LIN {X 0,Y 540.367,Z 1010.165,A -85,B 0,C 180,E1 3978.151,E2 3978.151} C_VEL
LIN {X 0,Y 538.15,Z 995.311,A -85,B 0,C 180,E1 3978.449,E2 3978.449} C_VEL
LIN {X 0,Y 536.475,Z 989.03,A -85,B 0,C 180,E1 3978.66,E2 3978.66} C_VEL
LIN {X 0,Y 536.148,Z 989.03,A -85,B 0,C 180,E1 3984.971,E2 3984.971} C_VEL
LIN {X 0,Y 536.089,Z 989.03,A -85,B 0,C 180,E1 3990.441,E2 3990.441} C_VEL
LIN {X 0,Y 536.003,Z 989.03,A -85,B 0,C 180,E1 3996.241,E2 3996.241} C_VEL
LIN {X 0,Y 535.964,Z 989.03,A -85,B 0,C 180,E1 4002.507,E2 4002.507} C_VEL
LIN {X 0,Y 536.056,Z 989.03,A -85,B 0,C 180,E1 4007.493,E2 4007.493} C_VEL
LIN {X 0,Y 536.117,Z 989.03,A -85,B 0,C 180,E1 4013.761,E2 4013.761} C_VEL
LIN {X 0,Y 536.077,Z 989.03,A -85,B 0,C 180,E1 4019.552,E2 4019.552} C_VEL
LIN {X 0,Y 536.133,Z 989.03,A -85,B 0,C 180,E1 4020.914,E2 4020.914} C_VEL
LIN {X 0,Y 544.829,Z 1011.912,A -85,B 0,C 180,E1 4021.779,E2 4021.779} C_VEL
LIN {X 0,Y 544.168,Z 1050.277,A -85,B 0,C 180,E1 4022.566,E2 4022.566} C_VEL
LIN {X 0,Y 543.022,Z 1087.066,A -85,B 0,C 180,E1 4023.969,E2 4023.969} C_VEL
LIN {X 0,Y 541.475,Z 1121.1,A -85,B 0,C 180,E1 4025.943,E2 4025.943} C_VEL
LIN {X 0,Y 539.972,Z 1152.521,A -85,B 0,C 180,E1 4028.483,E2 4028.483} C_VEL
LIN {X 0,Y 538.584,Z 1181.234,A -85,B 0,C 180,E1 4031.623,E2 4031.623} C_VEL
LIN {X 0,Y 537.575,Z 1204.956,A -85,B 0,C 180,E1 4035.155,E2 4035.155} C_VEL
LIN {X 0,Y 537.021,Z 1223.191,A -85,B 0,C 180,E1 4038.924,E2 4038.924} C_VEL
LIN {X 0,Y 536.82,Z 1235.502,A -85,B 0,C 180,E1 4042.73,E2 4042.73} C_VEL
LIN {X 0,Y 536.779,Z 1242.723,A -85,B 0,C 180,E1 4046.774,E2 4046.774} C_VEL
LIN {X 0,Y 536.69,Z 1244.497,A -85,B 0,C 180,E1 4049.997,E2 4049.997} C_VEL
LIN {X 0,Y 536.816,Z 1241.65,A -85,B 0,C 180,E1 4054.01,E2 4054.01} C_VEL
LIN {X 0,Y 536.89,Z 1233.07,A -85,B 0,C 180,E1 4058.076,E2 4058.076} C_VEL
LIN {X 0,Y 537.166,Z 1219.982,A -85,B 0,C 180,E1 4061.749,E2 4061.749} C_VEL
LIN {X 0,Y 537.78,Z 1200.841,A -85,B 0,C 180,E1 4065.458,E2 4065.458} C_VEL
LIN {X 0,Y 538.787,Z 1177.187,A -85,B 0,C 180,E1 4068.786,E2 4068.786} C_VEL
LIN {X 0,Y 540.151,Z 1149.395,A -85,B 0,C 180,E1 4071.717,E2 4071.717} C_VEL
LIN {X 0,Y 541.704,Z 1116.776,A -85,B 0,C 180,E1 4074.258,E2 4074.258} C_VEL
LIN {X 0,Y 543.1,Z 1082.588,A -85,B 0,C 180,E1 4076.148,E2 4076.148} C_VEL
LIN {X 0,Y 544.272,Z 1045.483,A -85,B 0,C 180,E1 4077.481,E2 4077.481} C_VEL
LIN {X 0,Y 544.242,Z 1008.876,A -85,B 0,C 180,E1 4078.209,E2 4078.209} C_VEL
LIN {X 0,Y 536.279,Z 989.03,A -85,B 0,C 180,E1 4079.036,E2 4079.036} C_VEL
LIN {X 0,Y 536.021,Z 989.03,A -85,B 0,C 180,E1 4085.277,E2 4085.277} C_VEL
LIN {X 0,Y 535.953,Z 989.03,A -85,B 0,C 180,E1 4090.522,E2 4090.522} C_VEL
LIN {X 0,Y 536.032,Z 989.03,A -85,B 0,C 180,E1 4097.046,E2 4097.046} C_VEL
LIN {X 0,Y 536.16,Z 989.03,A -85,B 0,C 180,E1 4102.001,E2 4102.001} C_VEL
LIN {X 0,Y 536.064,Z 989.03,A -85,B 0,C 180,E1 4107.669,E2 4107.669} C_VEL
LIN {X 0,Y 536.162,Z 989.03,A -85,B 0,C 180,E1 4113.238,E2 4113.238} C_VEL
LIN {X 0,Y 536.256,Z 989.03,A -85,B 0,C 180,E1 4118.544,E2 4118.544} C_VEL
LIN {X 0,Y 536.371,Z 989.03,A -85,B 0,C 180,E1 4123.661,E2 4123.661} C_VEL
LIN {X 0,Y 536.376,Z 989.03,A -85,B 0,C 180,E1 4128.643,E2 4128.643} C_VEL
LIN {X 0,Y 536.424,Z 989.03,A -85,B 0,C 180,E1 4133.54,E2 4133.54} C_VEL
LIN {X 0,Y 536.402,Z 989.03,A -85,B 0,C 180,E1 4138.388,E2 4138.388} C_VEL
LIN {X 0,Y 536.458,Z 989.03,A -85,B 0,C 180,E1 4143.225,E2 4143.225} C_VEL
LIN {X 0,Y 536.344,Z 989.03,A -85,B 0,C 180,E1 4148.087,E2 4148.087} C_VEL
LIN {X 0,Y 536.321,Z 989.03,A -85,B 0,C 180,E1 4153.008,E2 4153.008} C_VEL
LIN {X 0,Y 536.256,Z 989.03,A -85,B 0,C 180,E1 4158.031,E2 4158.031} C_VEL
LIN {X 0,Y 536.189,Z 989.03,A -85,B 0,C 180,E1 4163.203,E2 4163.203} C_VEL
LIN {X 0,Y 536.17,Z 989.03,A -85,B 0,C 180,E1 4166.745,E2 4166.745} C_VEL
LIN {X 0,Y 533.647,Z 989.03,A -85,B 0,C 180,E1 4168.125,E2 4168.125} C_VEL
LIN {X 0,Y 528.17,Z 989.03,A -85,B 0,C 180,E1 4170.192,E2 4170.192} C_VEL
LIN {X 0,Y 528.081,Z 989.03,A -85,B 0,C 180,E1 4170.431,E2 4170.431} C_VEL
LIN {X 0,Y 528.183,Z 989.03,A -85,B 0,C 180,E1 4176.877,E2 4176.877} C_VEL
LIN {X 0,Y 528.102,Z 989.03,A -85,B 0,C 180,E1 4182.021,E2 4182.021} C_VEL
LIN {X 0,Y 527.988,Z 989.03,A -85,B 0,C 180,E1 4187.993,E2 4187.993} C_VEL
LIN {X 0,Y 528.102,Z 989.11,A -85,B 0,C 180,E1 4193.2,E2 4193.2} C_VEL
LIN {X 0,Y 531.272,Z 996.761,A -85,B 0,C 180,E1 4194.015,E2 4194.015} C_VEL
LIN {X 0,Y 534.684,Z 1001.319,A -85,B 0,C 180,E1 4194.927,E2 4194.927} C_VEL
LIN {X 0,Y 536.379,Z 1002.647,A -85,B 0,C 180,E1 4195.518,E2 4195.518} C_VEL
LIN {X 0,Y 536.746,Z 1007.356,A -85,B 0,C 180,E1 4196.014,E2 4196.014} C_VEL
LIN {X 0,Y 540.769,Z 1015.949,A -85,B 0,C 180,E1 4196.435,E2 4196.435} C_VEL
LIN {X 0,Y 540.154,Z 1080.881,A -85,B 0,C 180,E1 4197.563,E2 4197.563} C_VEL
LIN {X 0,Y 538.764,Z 1119.195,A -85,B 0,C 180,E1 4198.853,E2 4198.853} C_VEL
LIN {X 0,Y 536.801,Z 1156.353,A -85,B 0,C 180,E1 4200.759,E2 4200.759} C_VEL
LIN {X 0,Y 534.581,Z 1192.701,A -85,B 0,C 180,E1 4203.38,E2 4203.38} C_VEL
LIN {X 0,Y 532.599,Z 1224.03,A -85,B 0,C 180,E1 4206.412,E2 4206.412} C_VEL
LIN {X 0,Y 530.966,Z 1251.131,A -85,B 0,C 180,E1 4209.821,E2 4209.821} C_VEL
LIN {X 0,Y 529.76,Z 1274.259,A -85,B 0,C 180,E1 4213.666,E2 4213.666} C_VEL
LIN {X 0,Y 529.131,Z 1292.024,A -85,B 0,C 180,E1 4217.652,E2 4217.652} C_VEL
LIN {X 0,Y 528.92,Z 1303.716,A -85,B 0,C 180,E1 4221.389,E2 4221.389} C_VEL
LIN {X 0,Y 528.753,Z 1310.987,A -85,B 0,C 180,E1 4225.092,E2 4225.092} C_VEL
LIN {X 0,Y 528.767,Z 1314.109,A -85,B 0,C 180,E1 4228.368,E2 4228.368} C_VEL
LIN {X 0,Y 528.742,Z 1313.363,A -85,B 0,C 180,E1 4232.755,E2 4232.755} C_VEL
LIN {X 0,Y 528.858,Z 1308.232,A -85,B 0,C 180,E1 4236.557,E2 4236.557} C_VEL
LIN {X 0,Y 528.957,Z 1298.391,A -85,B 0,C 180,E1 4240.489,E2 4240.489} C_VEL
LIN {X 0,Y 529.512,Z 1283.109,A -85,B 0,C 180,E1 4244.508,E2 4244.508} C_VEL
LIN {X 0,Y 530.409,Z 1262.353,A -85,B 0,C 180,E1 4248.456,E2 4248.456} C_VEL
LIN {X 0,Y 531.918,Z 1235.368,A -85,B 0,C 180,E1 4252.267,E2 4252.267} C_VEL
LIN {X 0,Y 533.841,Z 1204.625,A -85,B 0,C 180,E1 4255.566,E2 4255.566} C_VEL
LIN {X 0,Y 535.9,Z 1170.548,A -85,B 0,C 180,E1 4258.32,E2 4258.32} C_VEL
LIN {X 0,Y 538.097,Z 1132.34,A -85,B 0,C 180,E1 4260.554,E2 4260.554} C_VEL
LIN {X 0,Y 539.702,Z 1093.317,A -85,B 0,C 180,E1 4262.094,E2 4262.094} C_VEL
LIN {X 0,Y 540.821,Z 1051.141,A -85,B 0,C 180,E1 4263.013,E2 4263.013} C_VEL
LIN {X 0,Y 540.426,Z 1015.815,A -85,B 0,C 180,E1 4263.591,E2 4263.591} C_VEL
LIN {X 0,Y 535.954,Z 1006.21,A -85,B 0,C 180,E1 4264.108,E2 4264.108} C_VEL
LIN {X 0,Y 535.635,Z 1002.325,A -85,B 0,C 180,E1 4264.743,E2 4264.743} C_VEL
LIN {X 0,Y 531.269,Z 996.807,A -85,B 0,C 180,E1 4265.982,E2 4265.982} C_VEL
LIN {X 0,Y 528.163,Z 989.03,A -85,B 0,C 180,E1 4266.874,E2 4266.874} C_VEL
LIN {X 0,Y 528.107,Z 989.03,A -85,B 0,C 180,E1 4273.303,E2 4273.303} C_VEL
LIN {X 0,Y 527.998,Z 989.03,A -85,B 0,C 180,E1 4278.905,E2 4278.905} C_VEL
LIN {X 0,Y 528.146,Z 989.03,A -85,B 0,C 180,E1 4285.151,E2 4285.151} C_VEL
LIN {X 0,Y 528.268,Z 989.03,A -85,B 0,C 180,E1 4290.949,E2 4290.949} C_VEL
LIN {X 0,Y 528.254,Z 989.03,A -85,B 0,C 180,E1 4296.427,E2 4296.427} C_VEL
LIN {X 0,Y 528.435,Z 989.03,A -85,B 0,C 180,E1 4298.979,E2 4298.979} C_VEL
LIN {X 0,Y 533.189,Z 1007.897,A -85,B 0,C 180,E1 4299.451,E2 4299.451} C_VEL
LIN {X 0,Y 532.664,Z 1039.411,A -85,B 0,C 180,E1 4300.234,E2 4300.234} C_VEL
LIN {X 0,Y 531.883,Z 1068.952,A -85,B 0,C 180,E1 4301.602,E2 4301.602} C_VEL
LIN {X 0,Y 530.832,Z 1096.411,A -85,B 0,C 180,E1 4303.591,E2 4303.591} C_VEL
LIN {X 0,Y 529.996,Z 1120.443,A -85,B 0,C 180,E1 4306.117,E2 4306.117} C_VEL
LIN {X 0,Y 529.319,Z 1138.982,A -85,B 0,C 180,E1 4308.929,E2 4308.929} C_VEL
LIN {X 0,Y 529.04,Z 1153.365,A -85,B 0,C 180,E1 4312.213,E2 4312.213} C_VEL
LIN {X 0,Y 528.929,Z 1160.897,A -85,B 0,C 180,E1 4315.09,E2 4315.09} C_VEL
LIN {X 0,Y 528.892,Z 1164.4,A -85,B 0,C 180,E1 4318.365,E2 4318.365} C_VEL
LIN {X 0,Y 528.97,Z 1162.721,A -85,B 0,C 180,E1 4321.634,E2 4321.634} C_VEL
LIN {X 0,Y 529.046,Z 1155.841,A -85,B 0,C 180,E1 4324.908,E2 4324.908} C_VEL
LIN {X 0,Y 529.318,Z 1143.084,A -85,B 0,C 180,E1 4328.194,E2 4328.194} C_VEL
LIN {X 0,Y 529.855,Z 1124.21,A -85,B 0,C 180,E1 4331.293,E2 4331.293} C_VEL
LIN {X 0,Y 530.668,Z 1101.303,A -85,B 0,C 180,E1 4333.881,E2 4333.881} C_VEL
LIN {X 0,Y 531.712,Z 1073.59,A -85,B 0,C 180,E1 4336.02,E2 4336.02} C_VEL
LIN {X 0,Y 532.623,Z 1044.543,A -85,B 0,C 180,E1 4337.491,E2 4337.491} C_VEL
LIN {X 0,Y 533.002,Z 1013.899,A -85,B 0,C 180,E1 4338.358,E2 4338.358} C_VEL
LIN {X 0,Y 531.151,Z 998.292,A -85,B 0,C 180,E1 4338.674,E2 4338.674} C_VEL
LIN {X 0,Y 528.549,Z 989.03,A -85,B 0,C 180,E1 4338.974,E2 4338.974} C_VEL
LIN {X 0,Y 528.228,Z 989.03,A -85,B 0,C 180,E1 4345.371,E2 4345.371} C_VEL
LIN {X 0,Y 528.162,Z 989.03,A -85,B 0,C 180,E1 4350.995,E2 4350.995} C_VEL
LIN {X 0,Y 528.053,Z 989.03,A -85,B 0,C 180,E1 4356.876,E2 4356.876} C_VEL
LIN {X 0,Y 528.026,Z 989.03,A -85,B 0,C 180,E1 4363.302,E2 4363.302} C_VEL
LIN {X 0,Y 528.101,Z 989.03,A -85,B 0,C 180,E1 4368.907,E2 4368.907} C_VEL
LIN {X 0,Y 528.114,Z 989.03,A -85,B 0,C 180,E1 4375.142,E2 4375.142} C_VEL
LIN {X 0,Y 528.225,Z 989.03,A -85,B 0,C 180,E1 4380.452,E2 4380.452} C_VEL
LIN {X 0,Y 537.845,Z 1013.807,A -85,B 0,C 180,E1 4381.408,E2 4381.408} C_VEL
LIN {X 0,Y 537.092,Z 1052.408,A -85,B 0,C 180,E1 4382.24,E2 4382.24} C_VEL
LIN {X 0,Y 535.819,Z 1087.877,A -85,B 0,C 180,E1 4383.635,E2 4383.635} C_VEL
LIN {X 0,Y 534.065,Z 1122.589,A -85,B 0,C 180,E1 4385.699,E2 4385.699} C_VEL
LIN {X 0,Y 532.484,Z 1152.767,A -85,B 0,C 180,E1 4388.19,E2 4388.19} C_VEL
LIN {X 0,Y 530.958,Z 1181.231,A -85,B 0,C 180,E1 4391.349,E2 4391.349} C_VEL
LIN {X 0,Y 529.809,Z 1204.949,A -85,B 0,C 180,E1 4394.932,E2 4394.932} C_VEL
LIN {X 0,Y 529.166,Z 1222.052,A -85,B 0,C 180,E1 4398.482,E2 4398.482} C_VEL
LIN {X 0,Y 528.936,Z 1234.434,A -85,B 0,C 180,E1 4402.208,E2 4402.208} C_VEL
LIN {X 0,Y 528.876,Z 1241.749,A -85,B 0,C 180,E1 4405.906,E2 4405.906} C_VEL
LIN {X 0,Y 528.791,Z 1244.498,A -85,B 0,C 180,E1 4409.997,E2 4409.997} C_VEL
LIN {X 0,Y 528.914,Z 1241.626,A -85,B 0,C 180,E1 4414.087,E2 4414.087} C_VEL
LIN {X 0,Y 529.017,Z 1233.073,A -85,B 0,C 180,E1 4418.197,E2 4418.197} C_VEL
LIN {X 0,Y 529.307,Z 1219.987,A -85,B 0,C 180,E1 4421.926,E2 4421.926} C_VEL
LIN {X 0,Y 529.997,Z 1200.843,A -85,B 0,C 180,E1 4425.69,E2 4425.69} C_VEL
LIN {X 0,Y 531.133,Z 1177.19,A -85,B 0,C 180,E1 4429.068,E2 4429.068} C_VEL
LIN {X 0,Y 532.632,Z 1149.904,A -85,B 0,C 180,E1 4431.991,E2 4431.991} C_VEL
LIN {X 0,Y 534.319,Z 1118.432,A -85,B 0,C 180,E1 4434.504,E2 4434.504} C_VEL
LIN {X 0,Y 535.945,Z 1083.305,A -85,B 0,C 180,E1 4436.49,E2 4436.49} C_VEL
LIN {X 0,Y 537.23,Z 1046.617,A -85,B 0,C 180,E1 4437.839,E2 4437.839} C_VEL
LIN {X 0,Y 537.183,Z 1010.892,A -85,B 0,C 180,E1 4438.584,E2 4438.584} C_VEL
LIN {X 0,Y 528.354,Z 989.03,A -85,B 0,C 180,E1 4439.527,E2 4439.527} C_VEL
LIN {X 0,Y 528.134,Z 989.03,A -85,B 0,C 180,E1 4444.849,E2 4444.849} C_VEL
LIN {X 0,Y 527.987,Z 989.03,A -85,B 0,C 180,E1 4451.095,E2 4451.095} C_VEL
LIN {X 0,Y 528.082,Z 989.03,A -85,B 0,C 180,E1 4456.704,E2 4456.704} C_VEL
LIN {X 0,Y 528.179,Z 989.03,A -85,B 0,C 180,E1 4463.123,E2 4463.123} C_VEL
LIN {X 0,Y 528.144,Z 989.03,A -85,B 0,C 180,E1 4469.052,E2 4469.052} C_VEL
LIN {X 0,Y 528.256,Z 989.03,A -85,B 0,C 180,E1 4474.63,E2 4474.63} C_VEL
LIN {X 0,Y 528.46,Z 989.03,A -85,B 0,C 180,E1 4480.439,E2 4480.439} C_VEL
LIN {X 0,Y 528.566,Z 989.03,A -85,B 0,C 180,E1 4486.798,E2 4486.798} C_VEL
LIN {X 0,Y 528.506,Z 989.03,A -85,B 0,C 180,E1 4492.617,E2 4492.617} C_VEL
LIN {X 0,Y 528.53,Z 989.03,A -85,B 0,C 180,E1 4498.364,E2 4498.364} C_VEL
LIN {X 0,Y 528.565,Z 989.03,A -85,B 0,C 180,E1 4503.273,E2 4503.273} C_VEL
LIN {X 0,Y 528.447,Z 989.03,A -85,B 0,C 180,E1 4508.209,E2 4508.209} C_VEL
LIN {X 0,Y 528.361,Z 989.03,A -85,B 0,C 180,E1 4513.828,E2 4513.828} C_VEL
LIN {X 0,Y 528.38,Z 989.03,A -85,B 0,C 180,E1 4519.537,E2 4519.537} C_VEL
LIN {X 0,Y 528.256,Z 989.03,A -85,B 0,C 180,E1 4525.371,E2 4525.371} C_VEL
LIN {X 0,Y 528.081,Z 989.03,A -85,B 0,C 180,E1 4530.431,E2 4530.431} C_VEL
LIN {X 0,Y 525.572,Z 989.03,A -85,B 0,C 180,E1 4531.833,E2 4531.833} C_VEL
LIN {X 0,Y 520.182,Z 989.03,A -85,B 0,C 180,E1 4533.934,E2 4533.934} C_VEL
LIN {X 0,Y 520.079,Z 989.03,A -85,B 0,C 180,E1 4534.177,E2 4534.177} C_VEL
LIN {X 0,Y 520.247,Z 989.03,A -85,B 0,C 180,E1 4539.65,E2 4539.65} C_VEL
LIN {X 0,Y 520.119,Z 989.03,A -85,B 0,C 180,E1 4545.871,E2 4545.871} C_VEL
LIN {X 0,Y 520.114,Z 989.03,A -85,B 0,C 180,E1 4551.566,E2 4551.566} C_VEL
LIN {X 0,Y 520.17,Z 989.783,A -85,B 0,C 180,E1 4552.718,E2 4552.718} C_VEL
LIN {X 0,Y 525.693,Z 1002.215,A -85,B 0,C 180,E1 4553.879,E2 4553.879} C_VEL
LIN {X 0,Y 530.548,Z 1007.979,A -85,B 0,C 180,E1 4554.833,E2 4554.833} C_VEL
LIN {X 0,Y 532.192,Z 1010.059,A -85,B 0,C 180,E1 4555.311,E2 4555.311} C_VEL
LIN {X 0,Y 533.083,Z 1016.165,A -85,B 0,C 180,E1 4555.889,E2 4555.889} C_VEL
LIN {X 0,Y 534.339,Z 1021.051,A -85,B 0,C 180,E1 4556.058,E2 4556.058} C_VEL
LIN {X 0,Y 533.472,Z 1080.868,A -85,B 0,C 180,E1 4557.106,E2 4557.106} C_VEL
LIN {X 0,Y 531.885,Z 1119.703,A -85,B 0,C 180,E1 4558.428,E2 4558.428} C_VEL
LIN {X 0,Y 529.708,Z 1157.504,A -85,B 0,C 180,E1 4560.406,E2 4560.406} C_VEL
LIN {X 0,Y 527.331,Z 1192.696,A -85,B 0,C 180,E1 4562.984,E2 4562.984} C_VEL
LIN {X 0,Y 525.133,Z 1224.136,A -85,B 0,C 180,E1 4566.069,E2 4566.069} C_VEL
LIN {X 0,Y 523.361,Z 1251.4,A -85,B 0,C 180,E1 4569.555,E2 4569.555} C_VEL
LIN {X 0,Y 521.986,Z 1274.256,A -85,B 0,C 180,E1 4573.416,E2 4573.416} C_VEL
LIN {X 0,Y 521.315,Z 1292.027,A -85,B 0,C 180,E1 4577.464,E2 4577.464} C_VEL
LIN {X 0,Y 521.011,Z 1304.674,A -85,B 0,C 180,E1 4581.676,E2 4581.676} C_VEL
LIN {X 0,Y 520.858,Z 1310.99,A -85,B 0,C 180,E1 4585.017,E2 4585.017} C_VEL
LIN {X 0,Y 520.881,Z 1314.111,A -85,B 0,C 180,E1 4588.343,E2 4588.343} C_VEL
LIN {X 0,Y 520.994,Z 1314.106,A -85,B 0,C 180,E1 4591.663,E2 4591.663} C_VEL
LIN {X 0,Y 520.995,Z 1309.714,A -85,B 0,C 180,E1 4595.822,E2 4595.822} C_VEL
LIN {X 0,Y 521.078,Z 1300.086,A -85,B 0,C 180,E1 4600.076,E2 4600.076} C_VEL
LIN {X 0,Y 521.596,Z 1285.29,A -85,B 0,C 180,E1 4604.239,E2 4604.239} C_VEL
LIN {X 0,Y 522.64,Z 1263.63,A -85,B 0,C 180,E1 4608.522,E2 4608.522} C_VEL
LIN {X 0,Y 524.283,Z 1237.229,A -85,B 0,C 180,E1 4612.368,E2 4612.368} C_VEL
LIN {X 0,Y 526.335,Z 1207.184,A -85,B 0,C 180,E1 4615.703,E2 4615.703} C_VEL
LIN {X 0,Y 528.691,Z 1172.385,A -85,B 0,C 180,E1 4618.604,E2 4618.604} C_VEL
LIN {X 0,Y 531.069,Z 1135.145,A -85,B 0,C 180,E1 4620.855,E2 4620.855} C_VEL
LIN {X 0,Y 532.925,Z 1095.784,A -85,B 0,C 180,E1 4622.47,E2 4622.47} C_VEL
LIN {X 0,Y 534.211,Z 1054.855,A -85,B 0,C 180,E1 4623.415,E2 4623.415} C_VEL
LIN {X 0,Y 533.871,Z 1018.593,A -85,B 0,C 180,E1 4624.015,E2 4624.015} C_VEL
LIN {X 0,Y 532.004,Z 1013.248,A -85,B 0,C 180,E1 4624.395,E2 4624.395} C_VEL
LIN {X 0,Y 531.735,Z 1009.111,A -85,B 0,C 180,E1 4624.87,E2 4624.87} C_VEL
LIN {X 0,Y 526.81,Z 1004.036,A -85,B 0,C 180,E1 4625.903,E2 4625.903} C_VEL
LIN {X 0,Y 520.879,Z 992.093,A -85,B 0,C 180,E1 4626.991,E2 4626.991} C_VEL
LIN {X 0,Y 520.205,Z 989.03,A -85,B 0,C 180,E1 4627.305,E2 4627.305} C_VEL
LIN {X 0,Y 520.193,Z 989.03,A -85,B 0,C 180,E1 4633.516,E2 4633.516} C_VEL
LIN {X 0,Y 520.088,Z 989.03,A -85,B 0,C 180,E1 4638.978,E2 4638.978} C_VEL
LIN {X 0,Y 520.16,Z 989.03,A -85,B 0,C 180,E1 4644.536,E2 4644.536} C_VEL
LIN {X 0,Y 520.326,Z 989.03,A -85,B 0,C 180,E1 4650.473,E2 4650.473} C_VEL
LIN {X 0,Y 520.337,Z 989.03,A -85,B 0,C 180,E1 4656.046,E2 4656.046} C_VEL
LIN {X 0,Y 520.491,Z 989.03,A -85,B 0,C 180,E1 4658.665,E2 4658.665} C_VEL
LIN {X 0,Y 525.743,Z 1009.055,A -85,B 0,C 180,E1 4659.184,E2 4659.184} C_VEL
LIN {X 0,Y 525.084,Z 1041.909,A -85,B 0,C 180,E1 4660.046,E2 4660.046} C_VEL
LIN {X 0,Y 524.243,Z 1070.473,A -85,B 0,C 180,E1 4661.433,E2 4661.433} C_VEL
LIN {X 0,Y 523.103,Z 1097.393,A -85,B 0,C 180,E1 4663.45,E2 4663.45} C_VEL
LIN {X 0,Y 522.207,Z 1121,A -85,B 0,C 180,E1 4665.992,E2 4665.992} C_VEL
LIN {X 0,Y 521.472,Z 1139.75,A -85,B 0,C 180,E1 4668.928,E2 4668.928} C_VEL
LIN {X 0,Y 521.153,Z 1153.301,A -85,B 0,C 180,E1 4672.095,E2 4672.095} C_VEL
LIN {X 0,Y 521.03,Z 1160.859,A -85,B 0,C 180,E1 4675.015,E2 4675.015} C_VEL
LIN {X 0,Y 521.003,Z 1164.398,A -85,B 0,C 180,E1 4678.34,E2 4678.34} C_VEL
LIN {X 0,Y 521.08,Z 1162.737,A -85,B 0,C 180,E1 4681.659,E2 4681.659} C_VEL
LIN {X 0,Y 521.155,Z 1155.88,A -85,B 0,C 180,E1 4684.983,E2 4684.983} C_VEL
LIN {X 0,Y 521.464,Z 1143.161,A -85,B 0,C 180,E1 4688.319,E2 4688.319} C_VEL
LIN {X 0,Y 522.079,Z 1124.206,A -85,B 0,C 180,E1 4691.479,E2 4691.479} C_VEL
LIN {X 0,Y 522.959,Z 1101.684,A -85,B 0,C 180,E1 4694.071,E2 4694.071} C_VEL
LIN {X 0,Y 524.063,Z 1074.781,A -85,B 0,C 180,E1 4696.196,E2 4696.196} C_VEL
LIN {X 0,Y 525.067,Z 1046.246,A -85,B 0,C 180,E1 4697.699,E2 4697.699} C_VEL
LIN {X 0,Y 525.567,Z 1014.368,A -85,B 0,C 180,E1 4698.634,E2 4698.634} C_VEL
LIN {X 0,Y 523.494,Z 999.112,A -85,B 0,C 180,E1 4698.963,E2 4698.963} C_VEL
LIN {X 0,Y 520.599,Z 989.03,A -85,B 0,C 180,E1 4699.297,E2 4699.297} C_VEL
LIN {X 0,Y 520.266,Z 989.03,A -85,B 0,C 180,E1 4705.788,E2 4705.788} C_VEL
LIN {X 0,Y 520.231,Z 989.03,A -85,B 0,C 180,E1 4711.472,E2 4711.472} C_VEL
LIN {X 0,Y 520.054,Z 989.03,A -85,B 0,C 180,E1 4717.54,E2 4717.54} C_VEL
LIN {X 0,Y 520.122,Z 989.03,A -85,B 0,C 180,E1 4723.499,E2 4723.499} C_VEL
LIN {X 0,Y 520.196,Z 989.03,A -85,B 0,C 180,E1 4728.954,E2 4728.954} C_VEL
LIN {X 0,Y 520.166,Z 989.03,A -85,B 0,C 180,E1 4734.53,E2 4734.53} C_VEL
LIN {X 0,Y 520.283,Z 989.03,A -85,B 0,C 180,E1 4739.938,E2 4739.938} C_VEL
LIN {X 0,Y 530.83,Z 1015.719,A -85,B 0,C 180,E1 4741.023,E2 4741.023} C_VEL
LIN {X 0,Y 530.008,Z 1054.845,A -85,B 0,C 180,E1 4741.914,E2 4741.914} C_VEL
LIN {X 0,Y 528.572,Z 1090.66,A -85,B 0,C 180,E1 4743.398,E2 4743.398} C_VEL
LIN {X 0,Y 526.681,Z 1124.079,A -85,B 0,C 180,E1 4745.448,E2 4745.448} C_VEL
LIN {X 0,Y 524.801,Z 1156.107,A -85,B 0,C 180,E1 4748.185,E2 4748.185} C_VEL
LIN {X 0,Y 523.203,Z 1182.821,A -85,B 0,C 180,E1 4751.281,E2 4751.281} C_VEL
LIN {X 0,Y 521.99,Z 1206.129,A -85,B 0,C 180,E1 4754.916,E2 4754.916} C_VEL
LIN {X 0,Y 521.284,Z 1223.735,A -85,B 0,C 180,E1 4758.729,E2 4758.729} C_VEL
LIN {X 0,Y 521.048,Z 1235.5,A -85,B 0,C 180,E1 4762.508,E2 4762.508} C_VEL
LIN {X 0,Y 520.994,Z 1242.721,A -85,B 0,C 180,E1 4766.676,E2 4766.676} C_VEL
LIN {X 0,Y 520.897,Z 1244.498,A -85,B 0,C 180,E1 4769.997,E2 4769.997} C_VEL
LIN {X 0,Y 521.011,Z 1241.627,A -85,B 0,C 180,E1 4774.149,E2 4774.149} C_VEL
LIN {X 0,Y 521.135,Z 1233.075,A -85,B 0,C 180,E1 4778.322,E2 4778.322} C_VEL
LIN {X 0,Y 521.484,Z 1219.992,A -85,B 0,C 180,E1 4782.107,E2 4782.107} C_VEL
LIN {X 0,Y 522.223,Z 1200.845,A -85,B 0,C 180,E1 4785.93,E2 4785.93} C_VEL
LIN {X 0,Y 523.498,Z 1177.193,A -85,B 0,C 180,E1 4789.357,E2 4789.357} C_VEL
LIN {X 0,Y 525.292,Z 1148.415,A -85,B 0,C 180,E1 4792.462,E2 4792.462} C_VEL
LIN {X 0,Y 527.152,Z 1116.792,A -85,B 0,C 180,E1 4794.973,E2 4794.973} C_VEL
LIN {X 0,Y 528.847,Z 1082.445,A -85,B 0,C 180,E1 4796.916,E2 4796.916} C_VEL
LIN {X 0,Y 530.301,Z 1045.179,A -85,B 0,C 180,E1 4798.279,E2 4798.279} C_VEL
LIN {X 0,Y 530.31,Z 1013.247,A -85,B 0,C 180,E1 4798.957,E2 4798.957} C_VEL
LIN {X 0,Y 520.389,Z 989.03,A -85,B 0,C 180,E1 4799.993,E2 4799.993} C_VEL
LIN {X 0,Y 520.135,Z 989.03,A -85,B 0,C 180,E1 4805.68,E2 4805.68} C_VEL
LIN {X 0,Y 520.078,Z 989.03,A -85,B 0,C 180,E1 4811.86,E2 4811.86} C_VEL
LIN {X 0,Y 520.192,Z 989.03,A -85,B 0,C 180,E1 4818.151,E2 4818.151} C_VEL
LIN {X 0,Y 520.195,Z 989.03,A -85,B 0,C 180,E1 4824.312,E2 4824.312} C_VEL
LIN {X 0,Y 520.239,Z 989.03,A -85,B 0,C 180,E1 4830.476,E2 4830.476} C_VEL
LIN {X 0,Y 520.362,Z 989.03,A -85,B 0,C 180,E1 4836.048,E2 4836.048} C_VEL
LIN {X 0,Y 520.533,Z 989.03,A -85,B 0,C 180,E1 4841.406,E2 4841.406} C_VEL
LIN {X 0,Y 520.672,Z 989.03,A -85,B 0,C 180,E1 4846.595,E2 4846.595} C_VEL
LIN {X 0,Y 520.59,Z 989.03,A -85,B 0,C 180,E1 4852.617,E2 4852.617} C_VEL
LIN {X 0,Y 520.654,Z 989.03,A -85,B 0,C 180,E1 4858.34,E2 4858.34} C_VEL
LIN {X 0,Y 520.661,Z 989.03,A -85,B 0,C 180,E1 4863.323,E2 4863.323} C_VEL
LIN {X 0,Y 520.536,Z 989.03,A -85,B 0,C 180,E1 4868.334,E2 4868.334} C_VEL
LIN {X 0,Y 520.505,Z 989.03,A -85,B 0,C 180,E1 4873.41,E2 4873.41} C_VEL
LIN {X 0,Y 520.434,Z 989.03,A -85,B 0,C 180,E1 4878.599,E2 4878.599} C_VEL
LIN {X 0,Y 520.334,Z 989.03,A -85,B 0,C 180,E1 4883.954,E2 4883.954} C_VEL
LIN {X 0,Y 520.229,Z 989.03,A -85,B 0,C 180,E1 4889.544,E2 4889.544} C_VEL
LIN {X 0,Y 520.079,Z 989.03,A -85,B 0,C 180,E1 4894.177,E2 4894.177} C_VEL
LIN {X 0,Y 516.147,Z 989.03,A -85,B 0,C 180,E1 4896.063,E2 4896.063} C_VEL
LIN {X 0,Y 512.291,Z 989.03,A -85,B 0,C 180,E1 4897.978,E2 4897.978} C_VEL
LIN {X 0,Y 512.245,Z 989.03,A -85,B 0,C 180,E1 4902.651,E2 4902.651} C_VEL
LIN {X 0,Y 512.151,Z 989.03,A -85,B 0,C 180,E1 4907.44,E2 4907.44} C_VEL
LIN {X 0,Y 512.201,Z 989.374,A -85,B 0,C 180,E1 4912.146,E2 4912.146} C_VEL
LIN {X 0,Y 517.902,Z 1004.047,A -85,B 0,C 180,E1 4913.479,E2 4913.479} C_VEL
LIN {X 0,Y 524.083,Z 1012.79,A -85,B 0,C 180,E1 4914.467,E2 4914.467} C_VEL
LIN {X 0,Y 527.212,Z 1016.466,A -85,B 0,C 180,E1 4915.082,E2 4915.082} C_VEL
LIN {X 0,Y 527.708,Z 1021.249,A -85,B 0,C 180,E1 4915.567,E2 4915.567} C_VEL
LIN {X 0,Y 526.827,Z 1081.066,A -85,B 0,C 180,E1 4916.643,E2 4916.643} C_VEL
LIN {X 0,Y 525.09,Z 1119.695,A -85,B 0,C 180,E1 4917.972,E2 4917.972} C_VEL
LIN {X 0,Y 522.7,Z 1157.995,A -85,B 0,C 180,E1 4920.003,E2 4920.003} C_VEL
LIN {X 0,Y 520.014,Z 1193.968,A -85,B 0,C 180,E1 4922.689,E2 4922.689} C_VEL
LIN {X 0,Y 517.584,Z 1225.953,A -85,B 0,C 180,E1 4925.913,E2 4925.913} C_VEL
LIN {X 0,Y 515.534,Z 1253.935,A -85,B 0,C 180,E1 4929.619,E2 4929.619} C_VEL
LIN {X 0,Y 514.069,Z 1277.513,A -85,B 0,C 180,E1 4933.81,E2 4933.81} C_VEL
LIN {X 0,Y 513.403,Z 1293.568,A -85,B 0,C 180,E1 4937.699,E2 4937.699} C_VEL
LIN {X 0,Y 513.153,Z 1304.673,A -85,B 0,C 180,E1 4941.548,E2 4941.548} C_VEL
LIN {X 0,Y 512.968,Z 1310.993,A -85,B 0,C 180,E1 4944.94,E2 4944.94} C_VEL
LIN {X 0,Y 512.995,Z 1314.112,A -85,B 0,C 180,E1 4948.318,E2 4948.318} C_VEL
LIN {X 0,Y 513.104,Z 1314.108,A -85,B 0,C 180,E1 4951.689,E2 4951.689} C_VEL
LIN {X 0,Y 513.099,Z 1309.711,A -85,B 0,C 180,E1 4955.912,E2 4955.912} C_VEL
LIN {X 0,Y 513.208,Z 1300.266,A -85,B 0,C 180,E1 4960.165,E2 4960.165} C_VEL
LIN {X 0,Y 513.745,Z 1286.181,A -85,B 0,C 180,E1 4964.243,E2 4964.243} C_VEL
LIN {X 0,Y 514.766,Z 1266.306,A -85,B 0,C 180,E1 4968.331,E2 4968.331} C_VEL
LIN {X 0,Y 516.464,Z 1241.927,A -85,B 0,C 180,E1 4972.102,E2 4972.102} C_VEL
LIN {X 0,Y 518.756,Z 1210.818,A -85,B 0,C 180,E1 4975.724,E2 4975.724} C_VEL
LIN {X 0,Y 521.282,Z 1177.387,A -85,B 0,C 180,E1 4978.654,E2 4978.654} C_VEL
LIN {X 0,Y 523.884,Z 1140.473,A -85,B 0,C 180,E1 4981.02,E2 4981.02} C_VEL
LIN {X 0,Y 525.941,Z 1102.971,A -85,B 0,C 180,E1 4982.686,E2 4982.686} C_VEL
LIN {X 0,Y 527.448,Z 1065.41,A -85,B 0,C 180,E1 4983.703,E2 4983.703} C_VEL
LIN {X 0,Y 527.479,Z 1021.279,A -85,B 0,C 180,E1 4984.467,E2 4984.467} C_VEL
LIN {X 0,Y 526.241,Z 1014.664,A -85,B 0,C 180,E1 4985.18,E2 4985.18} C_VEL
LIN {X 0,Y 519.208,Z 1006.614,A -85,B 0,C 180,E1 4986.243,E2 4986.243} C_VEL
LIN {X 0,Y 513.052,Z 993.331,A -85,B 0,C 180,E1 4987.196,E2 4987.196} C_VEL
LIN {X 0,Y 512.295,Z 989.03,A -85,B 0,C 180,E1 4987.5,E2 4987.5} C_VEL
LIN {X 0,Y 512.27,Z 989.03,A -85,B 0,C 180,E1 4992.656,E2 4992.656} C_VEL
LIN {X 0,Y 512.179,Z 989.03,A -85,B 0,C 180,E1 4997.446,E2 4997.446} C_VEL
LIN {X 0,Y 512.199,Z 989.03,A -85,B 0,C 180,E1 5003.899,E2 5003.899} C_VEL
LIN {X 0,Y 512.371,Z 989.03,A -85,B 0,C 180,E1 5009.956,E2 5009.956} C_VEL
LIN {X 0,Y 512.423,Z 989.03,A -85,B 0,C 180,E1 5015.921,E2 5015.921} C_VEL
LIN {X 0,Y 512.565,Z 989.036,A -85,B 0,C 180,E1 5018.332,E2 5018.332} C_VEL
LIN {X 0,Y 518.331,Z 1010.908,A -85,B 0,C 180,E1 5018.914,E2 5018.914} C_VEL
LIN {X 0,Y 517.632,Z 1043.444,A -85,B 0,C 180,E1 5019.802,E2 5019.802} C_VEL
LIN {X 0,Y 516.593,Z 1071.906,A -85,B 0,C 180,E1 5021.258,E2 5021.258} C_VEL
LIN {X 0,Y 515.369,Z 1099.548,A -85,B 0,C 180,E1 5023.413,E2 5023.413} C_VEL
LIN {X 0,Y 514.398,Z 1121.981,A -85,B 0,C 180,E1 5025.923,E2 5025.923} C_VEL
LIN {X 0,Y 513.574,Z 1140.846,A -85,B 0,C 180,E1 5028.99,E2 5028.99} C_VEL
LIN {X 0,Y 513.311,Z 1154.655,A -85,B 0,C 180,E1 5032.398,E2 5032.398} C_VEL
LIN {X 0,Y 513.147,Z 1162.162,A -85,B 0,C 180,E1 5035.784,E2 5035.784} C_VEL
LIN {X 0,Y 513.117,Z 1164.396,A -85,B 0,C 180,E1 5038.315,E2 5038.315} C_VEL
LIN {X 0,Y 513.179,Z 1162.753,A -85,B 0,C 180,E1 5041.685,E2 5041.685} C_VEL
LIN {X 0,Y 513.271,Z 1155.918,A -85,B 0,C 180,E1 5045.059,E2 5045.059} C_VEL
LIN {X 0,Y 513.631,Z 1143.238,A -85,B 0,C 180,E1 5048.446,E2 5048.446} C_VEL
LIN {X 0,Y 514.248,Z 1125.052,A -85,B 0,C 180,E1 5051.549,E2 5051.549} C_VEL
LIN {X 0,Y 515.17,Z 1103.722,A -85,B 0,C 180,E1 5054.102,E2 5054.102} C_VEL
LIN {X 0,Y 516.333,Z 1078.214,A -85,B 0,C 180,E1 5056.227,E2 5056.227} C_VEL
LIN {X 0,Y 517.542,Z 1047.532,A -85,B 0,C 180,E1 5057.933,E2 5057.933} C_VEL
LIN {X 0,Y 518.194,Z 1017.287,A -85,B 0,C 180,E1 5058.878,E2 5058.878} C_VEL
LIN {X 0,Y 516.45,Z 1001.738,A -85,B 0,C 180,E1 5059.227,E2 5059.227} C_VEL
LIN {X 0,Y 512.662,Z 989.03,A -85,B 0,C 180,E1 5059.61,E2 5059.61} C_VEL
LIN {X 0,Y 512.343,Z 989.03,A -85,B 0,C 180,E1 5066.217,E2 5066.217} C_VEL
LIN {X 0,Y 512.308,Z 989.03,A -85,B 0,C 180,E1 5072.016,E2 5072.016} C_VEL
LIN {X 0,Y 512.138,Z 989.03,A -85,B 0,C 180,E1 5078.223,E2 5078.223} C_VEL
LIN {X 0,Y 512.239,Z 989.03,A -85,B 0,C 180,E1 5085.001,E2 5085.001} C_VEL
LIN {X 0,Y 512.304,Z 989.03,A -85,B 0,C 180,E1 5089.978,E2 5089.978} C_VEL
LIN {X 0,Y 512.211,Z 989.03,A -85,B 0,C 180,E1 5095.956,E2 5095.956} C_VEL
LIN {X 0,Y 512.393,Z 989.631,A -85,B 0,C 180,E1 5099.443,E2 5099.443} C_VEL
LIN {X 0,Y 524.021,Z 1018.676,A -85,B 0,C 180,E1 5100.649,E2 5100.649} C_VEL
LIN {X 0,Y 522.997,Z 1056.834,A -85,B 0,C 180,E1 5101.561,E2 5101.561} C_VEL
LIN {X 0,Y 521.396,Z 1091.635,A -85,B 0,C 180,E1 5103.052,E2 5103.052} C_VEL
LIN {X 0,Y 519.307,Z 1125.569,A -85,B 0,C 180,E1 5105.191,E2 5105.191} C_VEL
LIN {X 0,Y 517.283,Z 1156.784,A -85,B 0,C 180,E1 5107.925,E2 5107.925} C_VEL
LIN {X 0,Y 515.444,Z 1184.388,A -85,B 0,C 180,E1 5111.21,E2 5111.21} C_VEL
LIN {X 0,Y 514.134,Z 1207.679,A -85,B 0,C 180,E1 5114.967,E2 5114.967} C_VEL
LIN {X 0,Y 513.395,Z 1225.262,A -85,B 0,C 180,E1 5118.982,E2 5118.982} C_VEL
LIN {X 0,Y 513.183,Z 1235.498,A -85,B 0,C 180,E1 5122.393,E2 5122.393} C_VEL
LIN {X 0,Y 513.11,Z 1242.72,A -85,B 0,C 180,E1 5126.625,E2 5126.625} C_VEL
LIN {X 0,Y 513,Z 1244.498,A -85,B 0,C 180,E1 5129.997,E2 5129.997} C_VEL
LIN {X 0,Y 513.127,Z 1241.628,A -85,B 0,C 180,E1 5134.213,E2 5134.213} C_VEL
LIN {X 0,Y 513.269,Z 1233.076,A -85,B 0,C 180,E1 5138.45,E2 5138.45} C_VEL
LIN {X 0,Y 513.635,Z 1219.997,A -85,B 0,C 180,E1 5142.295,E2 5142.295} C_VEL
LIN {X 0,Y 514.469,Z 1200.846,A -85,B 0,C 180,E1 5146.177,E2 5146.177} C_VEL
LIN {X 0,Y 515.885,Z 1177.197,A -85,B 0,C 180,E1 5149.654,E2 5149.654} C_VEL
LIN {X 0,Y 517.777,Z 1149.181,A -85,B 0,C 180,E1 5152.73,E2 5152.73} C_VEL
LIN {X 0,Y 519.893,Z 1116.8,A -85,B 0,C 180,E1 5155.346,E2 5155.346} C_VEL
LIN {X 0,Y 521.89,Z 1081.182,A -85,B 0,C 180,E1 5157.379,E2 5157.379} C_VEL
LIN {X 0,Y 523.448,Z 1044.241,A -85,B 0,C 180,E1 5158.729,E2 5158.729} C_VEL
LIN {X 0,Y 523.491,Z 1015.651,A -85,B 0,C 180,E1 5159.341,E2 5159.341} C_VEL
LIN {X 0,Y 512.453,Z 989.03,A -85,B 0,C 180,E1 5160.518,E2 5160.518} C_VEL
LIN {X 0,Y 512.193,Z 989.03,A -85,B 0,C 180,E1 5166.1,E2 5166.1} C_VEL
LIN {X 0,Y 512.149,Z 989.03,A -85,B 0,C 180,E1 5172.56,E2 5172.56} C_VEL
LIN {X 0,Y 512.247,Z 989.03,A -85,B 0,C 180,E1 5177.428,E2 5177.428} C_VEL
LIN {X 0,Y 512.292,Z 989.03,A -85,B 0,C 180,E1 5182.682,E2 5182.682} C_VEL
LIN {X 0,Y 512.288,Z 989.03,A -85,B 0,C 180,E1 5188.671,E2 5188.671} C_VEL
LIN {X 0,Y 512.367,Z 989.03,A -85,B 0,C 180,E1 5193.784,E2 5193.784} C_VEL
LIN {X 0,Y 512.556,Z 989.03,A -85,B 0,C 180,E1 5199.313,E2 5199.313} C_VEL
LIN {X 0,Y 512.677,Z 989.03,A -85,B 0,C 180,E1 5204.64,E2 5204.64} C_VEL
LIN {X 0,Y 512.705,Z 989.03,A -85,B 0,C 180,E1 5209.829,E2 5209.829} C_VEL
LIN {X 0,Y 512.814,Z 989.03,A -85,B 0,C 180,E1 5214.936,E2 5214.936} C_VEL
LIN {X 0,Y 513.015,Z 989.03,A -85,B 0,C 180,E1 5221.686,E2 5221.686} C_VEL
LIN {X 0,Y 512.808,Z 989.03,A -85,B 0,C 180,E1 5226.76,E2 5226.76} C_VEL
LIN {X 0,Y 512.635,Z 989.03,A -85,B 0,C 180,E1 5231.891,E2 5231.891} C_VEL
LIN {X 0,Y 512.548,Z 989.03,A -85,B 0,C 180,E1 5237.122,E2 5237.122} C_VEL
LIN {X 0,Y 512.431,Z 989.03,A -85,B 0,C 180,E1 5242.508,E2 5242.508} C_VEL
LIN {X 0,Y 512.349,Z 989.03,A -85,B 0,C 180,E1 5248.114,E2 5248.114} C_VEL
LIN {X 0,Y 512.191,Z 989.03,A -85,B 0,C 180,E1 5254.422,E2 5254.422} C_VEL
LIN {X 0,Y 512.291,Z 989.03,A -85,B 0,C 180,E1 5257.978,E2 5257.978} C_VEL
LIN {X 0,Y 509.812,Z 989.03,A -85,B 0,C 180,E1 5259.408,E2 5259.408} C_VEL
LIN {X 0,Y 504.248,Z 989.03,A -85,B 0,C 180,E1 5261.798,E2 5261.798} C_VEL
LIN {X 0,Y 504.172,Z 989.03,A -85,B 0,C 180,E1 5266.499,E2 5266.499} C_VEL
LIN {X 0,Y 504.303,Z 989.45,A -85,B 0,C 180,E1 5271.59,E2 5271.59} C_VEL
LIN {X 0,Y 511.305,Z 1008.26,A -85,B 0,C 180,E1 5273.313,E2 5273.313} C_VEL
LIN {X 0,Y 521.567,Z 1022.856,A -85,B 0,C 180,E1 5274.95,E2 5274.95} C_VEL
LIN {X 0,Y 521.211,Z 1029.379,A -85,B 0,C 180,E1 5275.218,E2 5275.218} C_VEL
LIN {X 0,Y 520.176,Z 1082.446,A -85,B 0,C 180,E1 5276.199,E2 5276.199} C_VEL
LIN {X 0,Y 518.327,Z 1120.287,A -85,B 0,C 180,E1 5277.532,E2 5277.532} C_VEL
LIN {X 0,Y 515.728,Z 1157.99,A -85,B 0,C 180,E1 5279.555,E2 5279.555} C_VEL
LIN {X 0,Y 512.877,Z 1193.65,A -85,B 0,C 180,E1 5282.247,E2 5282.247} C_VEL
LIN {X 0,Y 510.16,Z 1225.947,A -85,B 0,C 180,E1 5285.54,E2 5285.54} C_VEL
LIN {X 0,Y 507.947,Z 1253.93,A -85,B 0,C 180,E1 5289.3,E2 5289.3} C_VEL
LIN {X 0,Y 506.33,Z 1277.511,A -85,B 0,C 180,E1 5293.556,E2 5293.556} C_VEL
LIN {X 0,Y 505.572,Z 1293.572,A -85,B 0,C 180,E1 5297.506,E2 5297.506} C_VEL
LIN {X 0,Y 505.261,Z 1304.672,A -85,B 0,C 180,E1 5301.415,E2 5301.415} C_VEL
LIN {X 0,Y 505.075,Z 1310.995,A -85,B 0,C 180,E1 5304.861,E2 5304.861} C_VEL
LIN {X 0,Y 505.093,Z 1314.113,A -85,B 0,C 180,E1 5308.291,E2 5308.291} C_VEL
LIN {X 0,Y 505.197,Z 1314.109,A -85,B 0,C 180,E1 5311.715,E2 5311.715} C_VEL
LIN {X 0,Y 505.208,Z 1309.707,A -85,B 0,C 180,E1 5316.004,E2 5316.004} C_VEL
LIN {X 0,Y 505.325,Z 1300.264,A -85,B 0,C 180,E1 5320.325,E2 5320.325} C_VEL
LIN {X 0,Y 505.944,Z 1286.184,A -85,B 0,C 180,E1 5324.468,E2 5324.468} C_VEL
LIN {X 0,Y 507.116,Z 1265.818,A -85,B 0,C 180,E1 5328.706,E2 5328.706} C_VEL
LIN {X 0,Y 509.047,Z 1240.252,A -85,B 0,C 180,E1 5332.671,E2 5332.671} C_VEL
LIN {X 0,Y 511.66,Z 1208.327,A -85,B 0,C 180,E1 5336.379,E2 5336.379} C_VEL
LIN {X 0,Y 514.423,Z 1174.423,A -85,B 0,C 180,E1 5339.313,E2 5339.313} C_VEL
LIN {X 0,Y 517.284,Z 1136.744,A -85,B 0,C 180,E1 5341.679,E2 5341.679} C_VEL
LIN {X 0,Y 519.501,Z 1097.276,A -85,B 0,C 180,E1 5343.36,E2 5343.36} C_VEL
LIN {X 0,Y 521.051,Z 1056.927,A -85,B 0,C 180,E1 5344.337,E2 5344.337} C_VEL
LIN {X 0,Y 521.517,Z 1024.251,A -85,B 0,C 180,E1 5344.955,E2 5344.955} C_VEL
LIN {X 0,Y 519.034,Z 1018.874,A -85,B 0,C 180,E1 5345.509,E2 5345.509} C_VEL
LIN {X 0,Y 509.849,Z 1006.242,A -85,B 0,C 180,E1 5346.602,E2 5346.602} C_VEL
LIN {X 0,Y 504.756,Z 991.381,A -85,B 0,C 180,E1 5347.63,E2 5347.63} C_VEL
LIN {X 0,Y 504.387,Z 989.03,A -85,B 0,C 180,E1 5347.833,E2 5347.833} C_VEL
LIN {X 0,Y 504.264,Z 989.03,A -85,B 0,C 180,E1 5354.096,E2 5354.096} C_VEL
LIN {X 0,Y 504.182,Z 989.03,A -85,B 0,C 180,E1 5358.82,E2 5358.82} C_VEL
LIN {X 0,Y 504.345,Z 989.03,A -85,B 0,C 180,E1 5365.357,E2 5365.357} C_VEL
LIN {X 0,Y 504.421,Z 989.03,A -85,B 0,C 180,E1 5371.404,E2 5371.404} C_VEL
LIN {X 0,Y 504.657,Z 989.564,A -85,B 0,C 180,E1 5377.978,E2 5377.978} C_VEL
LIN {X 0,Y 510.953,Z 1011.632,A -85,B 0,C 180,E1 5378.608,E2 5378.608} C_VEL
LIN {X 0,Y 510.34,Z 1042.996,A -85,B 0,C 180,E1 5379.444,E2 5379.444} C_VEL
LIN {X 0,Y 509.369,Z 1071.479,A -85,B 0,C 180,E1 5380.87,E2 5380.87} C_VEL
LIN {X 0,Y 507.896,Z 1097.948,A -85,B 0,C 180,E1 5382.939,E2 5382.939} C_VEL
LIN {X 0,Y 506.671,Z 1121.034,A -85,B 0,C 180,E1 5385.59,E2 5385.59} C_VEL
LIN {X 0,Y 505.793,Z 1139.674,A -85,B 0,C 180,E1 5388.6,E2 5388.6} C_VEL
LIN {X 0,Y 505.416,Z 1153.174,A -85,B 0,C 180,E1 5391.847,E2 5391.847} C_VEL
LIN {X 0,Y 505.261,Z 1160.78,A -85,B 0,C 180,E1 5394.859,E2 5394.859} C_VEL
LIN {X 0,Y 505.215,Z 1164.395,A -85,B 0,C 180,E1 5398.288,E2 5398.288} C_VEL
LIN {X 0,Y 505.279,Z 1162.769,A -85,B 0,C 180,E1 5401.711,E2 5401.711} C_VEL
LIN {X 0,Y 505.381,Z 1155.957,A -85,B 0,C 180,E1 5405.139,E2 5405.139} C_VEL
LIN {X 0,Y 505.765,Z 1143.316,A -85,B 0,C 180,E1 5408.579,E2 5408.579} C_VEL
LIN {X 0,Y 506.481,Z 1124.546,A -85,B 0,C 180,E1 5411.819,E2 5411.819} C_VEL
LIN {X 0,Y 507.657,Z 1101.906,A -85,B 0,C 180,E1 5414.554,E2 5414.554} C_VEL
LIN {X 0,Y 509.074,Z 1074.541,A -85,B 0,C 180,E1 5416.798,E2 5416.798} C_VEL
LIN {X 0,Y 510.211,Z 1046.555,A -85,B 0,C 180,E1 5418.299,E2 5418.299} C_VEL
LIN {X 0,Y 510.786,Z 1015.326,A -85,B 0,C 180,E1 5419.233,E2 5419.233} C_VEL
LIN {X 0,Y 508.938,Z 1003,A -85,B 0,C 180,E1 5419.531,E2 5419.531} C_VEL
LIN {X 0,Y 504.702,Z 989.03,A -85,B 0,C 180,E1 5420,E2 5420} C_VEL
LIN {X 0,Y 504.398,Z 989.03,A -85,B 0,C 180,E1 5426.662,E2 5426.662} C_VEL
LIN {X 0,Y 504.307,Z 989.03,A -85,B 0,C 180,E1 5433.08,E2 5433.08} C_VEL
LIN {X 0,Y 504.197,Z 989.03,A -85,B 0,C 180,E1 5438.937,E2 5438.937} C_VEL
LIN {X 0,Y 504.242,Z 989.03,A -85,B 0,C 180,E1 5444.085,E2 5444.085} C_VEL
LIN {X 0,Y 504.285,Z 989.03,A -85,B 0,C 180,E1 5448.822,E2 5448.822} C_VEL
LIN {X 0,Y 504.396,Z 989.03,A -85,B 0,C 180,E1 5453.874,E2 5453.874} C_VEL
LIN {X 0,Y 504.424,Z 989.03,A -85,B 0,C 180,E1 5458.859,E2 5458.859} C_VEL
LIN {X 0,Y 517.147,Z 1021.217,A -85,B 0,C 180,E1 5460.256,E2 5460.256} C_VEL
LIN {X 0,Y 516.041,Z 1058.44,A -85,B 0,C 180,E1 5461.184,E2 5461.184} C_VEL
LIN {X 0,Y 514.316,Z 1093.202,A -85,B 0,C 180,E1 5462.709,E2 5462.709} C_VEL
LIN {X 0,Y 512.055,Z 1125.921,A -85,B 0,C 180,E1 5464.826,E2 5464.826} C_VEL
LIN {X 0,Y 509.736,Z 1157.908,A -85,B 0,C 180,E1 5467.706,E2 5467.706} C_VEL
LIN {X 0,Y 507.822,Z 1184.38,A -85,B 0,C 180,E1 5470.917,E2 5470.917} C_VEL
LIN {X 0,Y 506.373,Z 1207.464,A -85,B 0,C 180,E1 5474.69,E2 5474.69} C_VEL
LIN {X 0,Y 505.583,Z 1223.732,A -85,B 0,C 180,E1 5478.374,E2 5478.374} C_VEL
LIN {X 0,Y 505.288,Z 1235.497,A -85,B 0,C 180,E1 5482.273,E2 5482.273} C_VEL
LIN {X 0,Y 505.205,Z 1242.719,A -85,B 0,C 180,E1 5486.572,E2 5486.572} C_VEL
LIN {X 0,Y 505.1,Z 1244.498,A -85,B 0,C 180,E1 5489.997,E2 5489.997} C_VEL
LIN {X 0,Y 505.236,Z 1241.629,A -85,B 0,C 180,E1 5494.279,E2 5494.279} C_VEL
LIN {X 0,Y 505.378,Z 1233.078,A -85,B 0,C 180,E1 5498.583,E2 5498.583} C_VEL
LIN {X 0,Y 505.809,Z 1220,A -85,B 0,C 180,E1 5502.488,E2 5502.488} C_VEL
LIN {X 0,Y 506.716,Z 1200.848,A -85,B 0,C 180,E1 5506.431,E2 5506.431} C_VEL
LIN {X 0,Y 508.272,Z 1177.2,A -85,B 0,C 180,E1 5509.961,E2 5509.961} C_VEL
LIN {X 0,Y 510.395,Z 1148.417,A -85,B 0,C 180,E1 5513.156,E2 5513.156} C_VEL
LIN {X 0,Y 512.836,Z 1115.541,A -85,B 0,C 180,E1 5515.836,E2 5515.836} C_VEL
LIN {X 0,Y 514.902,Z 1081.752,A -85,B 0,C 180,E1 5517.783,E2 5517.783} C_VEL
LIN {X 0,Y 516.553,Z 1044.735,A -85,B 0,C 180,E1 5519.15,E2 5519.15} C_VEL
LIN {X 0,Y 516.56,Z 1017.689,A -85,B 0,C 180,E1 5519.749,E2 5519.749} C_VEL
LIN {X 0,Y 504.516,Z 989.03,A -85,B 0,C 180,E1 5521.076,E2 5521.076} C_VEL
LIN {X 0,Y 504.249,Z 989.03,A -85,B 0,C 180,E1 5526.761,E2 5526.761} C_VEL
LIN {X 0,Y 504.169,Z 989.03,A -85,B 0,C 180,E1 5533.501,E2 5533.501} C_VEL
LIN {X 0,Y 504.296,Z 989.03,A -85,B 0,C 180,E1 5538.832,E2 5538.832} C_VEL
LIN {X 0,Y 504.321,Z 989.03,A -85,B 0,C 180,E1 5545.356,E2 5545.356} C_VEL
LIN {X 0,Y 504.371,Z 989.03,A -85,B 0,C 180,E1 5551.401,E2 5551.401} C_VEL
LIN {X 0,Y 504.53,Z 989.03,A -85,B 0,C 180,E1 5557.12,E2 5557.12} C_VEL
LIN {X 0,Y 504.744,Z 989.03,A -85,B 0,C 180,E1 5563.069,E2 5563.069} C_VEL
LIN {X 0,Y 504.75,Z 989.03,A -85,B 0,C 180,E1 5567.921,E2 5567.921} C_VEL
LIN {X 0,Y 504.806,Z 989.03,A -85,B 0,C 180,E1 5573.133,E2 5573.133} C_VEL
LIN {X 0,Y 504.869,Z 989.03,A -85,B 0,C 180,E1 5578.288,E2 5578.288} C_VEL
LIN {X 0,Y 504.86,Z 989.03,A -85,B 0,C 180,E1 5583.427,E2 5583.427} C_VEL
LIN {X 0,Y 504.708,Z 989.03,A -85,B 0,C 180,E1 5589.381,E2 5589.381} C_VEL
LIN {X 0,Y 504.624,Z 989.03,A -85,B 0,C 180,E1 5595.612,E2 5595.612} C_VEL
LIN {X 0,Y 504.517,Z 989.03,A -85,B 0,C 180,E1 5602.001,E2 5602.001} C_VEL
LIN {X 0,Y 504.442,Z 989.03,A -85,B 0,C 180,E1 5606.66,E2 5606.66} C_VEL
LIN {X 0,Y 504.249,Z 989.03,A -85,B 0,C 180,E1 5613.082,E2 5613.082} C_VEL
LIN {X 0,Y 504.363,Z 989.03,A -85,B 0,C 180,E1 5618.935,E2 5618.935} C_VEL
LIN {X 0,Y 504.248,Z 989.03,A -85,B 0,C 180,E1 5621.798,E2 5621.798} C_VEL
LIN {X 0,Y 500.27,Z 989.03,A -85,B 0,C 180,E1 5623.746,E2 5623.746} C_VEL
LIN {X 0,Y 496.293,Z 989.03,A -85,B 0,C 180,E1 5625.724,E2 5625.724} C_VEL
LIN {X 0,Y 496.364,Z 989.674,A -85,B 0,C 180,E1 5631.03,E2 5631.03} C_VEL
LIN {X 0,Y 504.886,Z 1012.734,A -85,B 0,C 180,E1 5633.18,E2 5633.18} C_VEL
LIN {X 0,Y 514.696,Z 1026.091,A -85,B 0,C 180,E1 5634.674,E2 5634.674} C_VEL
LIN {X 0,Y 513.665,Z 1081.088,A -85,B 0,C 180,E1 5635.674,E2 5635.674} C_VEL
LIN {X 0,Y 511.669,Z 1119.042,A -85,B 0,C 180,E1 5636.995,E2 5636.995} C_VEL
LIN {X 0,Y 508.827,Z 1157.51,A -85,B 0,C 180,E1 5639.063,E2 5639.063} C_VEL
LIN {X 0,Y 505.756,Z 1193.211,A -85,B 0,C 180,E1 5641.78,E2 5641.78} C_VEL
LIN {X 0,Y 502.892,Z 1224.701,A -85,B 0,C 180,E1 5645.01,E2 5645.01} C_VEL
LIN {X 0,Y 500.448,Z 1252.78,A -85,B 0,C 180,E1 5648.79,E2 5648.79} C_VEL
LIN {X 0,Y 498.638,Z 1276.422,A -85,B 0,C 180,E1 5653.069,E2 5653.069} C_VEL
LIN {X 0,Y 497.743,Z 1293.574,A -85,B 0,C 180,E1 5657.306,E2 5657.306} C_VEL
LIN {X 0,Y 497.386,Z 1304.671,A -85,B 0,C 180,E1 5661.278,E2 5661.278} C_VEL
LIN {X 0,Y 497.184,Z 1310.998,A -85,B 0,C 180,E1 5664.779,E2 5664.779} C_VEL
LIN {X 0,Y 497.214,Z 1314.113,A -85,B 0,C 180,E1 5668.264,E2 5668.264} C_VEL
LIN {X 0,Y 497.292,Z 1314.11,A -85,B 0,C 180,E1 5671.742,E2 5671.742} C_VEL
LIN {X 0,Y 497.33,Z 1309.703,A -85,B 0,C 180,E1 5676.1,E2 5676.1} C_VEL
LIN {X 0,Y 497.442,Z 1300.261,A -85,B 0,C 180,E1 5680.491,E2 5680.491} C_VEL
LIN {X 0,Y 498.158,Z 1285.652,A -85,B 0,C 180,E1 5684.835,E2 5684.835} C_VEL
LIN {X 0,Y 499.503,Z 1264.843,A -85,B 0,C 180,E1 5689.184,E2 5689.184} C_VEL
LIN {X 0,Y 501.514,Z 1240.247,A -85,B 0,C 180,E1 5693.031,E2 5693.031} C_VEL
LIN {X 0,Y 504.286,Z 1209.4,A -85,B 0,C 180,E1 5696.675,E2 5696.675} C_VEL
LIN {X 0,Y 507.279,Z 1175.898,A -85,B 0,C 180,E1 5699.645,E2 5699.645} C_VEL
LIN {X 0,Y 510.324,Z 1138.974,A -85,B 0,C 180,E1 5702.029,E2 5702.029} C_VEL
LIN {X 0,Y 512.723,Z 1100.663,A -85,B 0,C 180,E1 5703.729,E2 5703.729} C_VEL
LIN {X 0,Y 514.378,Z 1062.135,A -85,B 0,C 180,E1 5704.734,E2 5704.734} C_VEL
LIN {X 0,Y 514.311,Z 1025.957,A -85,B 0,C 180,E1 5705.341,E2 5705.341} C_VEL
LIN {X 0,Y 502.329,Z 1009.053,A -85,B 0,C 180,E1 5706.73,E2 5706.73} C_VEL
LIN {X 0,Y 496.573,Z 989.894,A -85,B 0,C 180,E1 5708.049,E2 5708.049} C_VEL
LIN {X 0,Y 496.451,Z 989.03,A -85,B 0,C 180,E1 5708.699,E2 5708.699} C_VEL
LIN {X 0,Y 496.347,Z 989.03,A -85,B 0,C 180,E1 5714.373,E2 5714.373} C_VEL
LIN {X 0,Y 496.212,Z 989.03,A -85,B 0,C 180,E1 5720.313,E2 5720.313} C_VEL
LIN {X 0,Y 496.465,Z 989.03,A -85,B 0,C 180,E1 5726.832,E2 5726.832} C_VEL
LIN {X 0,Y 496.46,Z 989.03,A -85,B 0,C 180,E1 5732.876,E2 5732.876} C_VEL
LIN {X 0,Y 496.725,Z 989.221,A -85,B 0,C 180,E1 5737.595,E2 5737.595} C_VEL
LIN {X 0,Y 503.602,Z 1013.653,A -85,B 0,C 180,E1 5738.319,E2 5738.319} C_VEL
LIN {X 0,Y 502.974,Z 1045.481,A -85,B 0,C 180,E1 5739.187,E2 5739.187} C_VEL
LIN {X 0,Y 501.863,Z 1074.433,A -85,B 0,C 180,E1 5740.686,E2 5740.686} C_VEL
LIN {X 0,Y 500.434,Z 1100.474,A -85,B 0,C 180,E1 5742.79,E2 5742.79} C_VEL
LIN {X 0,Y 499.127,Z 1123.084,A -85,B 0,C 180,E1 5745.458,E2 5745.458} C_VEL
LIN {X 0,Y 498.007,Z 1141.349,A -85,B 0,C 180,E1 5748.641,E2 5748.641} C_VEL
LIN {X 0,Y 497.518,Z 1154.559,A -85,B 0,C 180,E1 5752.155,E2 5752.155} C_VEL
LIN {X 0,Y 497.364,Z 1162.107,A -85,B 0,C 180,E1 5755.65,E2 5755.65} C_VEL
LIN {X 0,Y 497.324,Z 1164.393,A -85,B 0,C 180,E1 5758.261,E2 5758.261} C_VEL
LIN {X 0,Y 497.406,Z 1162.785,A -85,B 0,C 180,E1 5761.738,E2 5761.738} C_VEL
LIN {X 0,Y 497.514,Z 1155.996,A -85,B 0,C 180,E1 5765.22,E2 5765.22} C_VEL
LIN {X 0,Y 497.938,Z 1143.702,A -85,B 0,C 180,E1 5768.715,E2 5768.715} C_VEL
LIN {X 0,Y 498.806,Z 1125.583,A -85,B 0,C 180,E1 5772.003,E2 5772.003} C_VEL
LIN {X 0,Y 500.075,Z 1103.498,A -85,B 0,C 180,E1 5774.737,E2 5774.737} C_VEL
LIN {X 0,Y 501.531,Z 1077.317,A -85,B 0,C 180,E1 5776.945,E2 5776.945} C_VEL
LIN {X 0,Y 502.799,Z 1048.171,A -85,B 0,C 180,E1 5778.562,E2 5778.562} C_VEL
LIN {X 0,Y 503.44,Z 1016.54,A -85,B 0,C 180,E1 5779.535,E2 5779.535} C_VEL
LIN {X 0,Y 501.605,Z 1004.605,A -85,B 0,C 180,E1 5779.831,E2 5779.831} C_VEL
LIN {X 0,Y 496.811,Z 989.03,A -85,B 0,C 180,E1 5780.373,E2 5780.373} C_VEL
LIN {X 0,Y 496.436,Z 989.03,A -85,B 0,C 180,E1 5787.125,E2 5787.125} C_VEL
LIN {X 0,Y 496.396,Z 989.03,A -85,B 0,C 180,E1 5793.172,E2 5793.172} C_VEL
LIN {X 0,Y 496.204,Z 989.03,A -85,B 0,C 180,E1 5799.687,E2 5799.687} C_VEL
LIN {X 0,Y 496.358,Z 989.03,A -85,B 0,C 180,E1 5805.628,E2 5805.628} C_VEL
LIN {X 0,Y 496.406,Z 989.03,A -85,B 0,C 180,E1 5812.216,E2 5812.216} C_VEL
LIN {X 0,Y 496.465,Z 989.03,A -85,B 0,C 180,E1 5818.322,E2 5818.322} C_VEL
LIN {X 0,Y 510.317,Z 1023.447,A -85,B 0,C 180,E1 5819.851,E2 5819.851} C_VEL
LIN {X 0,Y 509.139,Z 1059.594,A -85,B 0,C 180,E1 5820.781,E2 5820.781} C_VEL
LIN {X 0,Y 507.293,Z 1093.751,A -85,B 0,C 180,E1 5822.299,E2 5822.299} C_VEL
LIN {X 0,Y 504.866,Z 1126.76,A -85,B 0,C 180,E1 5824.464,E2 5824.464} C_VEL
LIN {X 0,Y 502.303,Z 1158.126,A -85,B 0,C 180,E1 5827.358,E2 5827.358} C_VEL
LIN {X 0,Y 500.029,Z 1186.618,A -85,B 0,C 180,E1 5830.934,E2 5830.934} C_VEL
LIN {X 0,Y 498.482,Z 1209.317,A -85,B 0,C 180,E1 5834.823,E2 5834.823} C_VEL
LIN {X 0,Y 497.688,Z 1225.254,A -85,B 0,C 180,E1 5838.63,E2 5838.63} C_VEL
LIN {X 0,Y 497.405,Z 1235.496,A -85,B 0,C 180,E1 5842.15,E2 5842.15} C_VEL
LIN {X 0,Y 497.327,Z 1242.718,A -85,B 0,C 180,E1 5846.517,E2 5846.517} C_VEL
LIN {X 0,Y 497.227,Z 1244.498,A -85,B 0,C 180,E1 5849.997,E2 5849.997} C_VEL
LIN {X 0,Y 497.333,Z 1241.63,A -85,B 0,C 180,E1 5854.347,E2 5854.347} C_VEL
LIN {X 0,Y 497.489,Z 1233.079,A -85,B 0,C 180,E1 5858.72,E2 5858.72} C_VEL
LIN {X 0,Y 497.998,Z 1220.001,A -85,B 0,C 180,E1 5862.688,E2 5862.688} C_VEL
LIN {X 0,Y 498.967,Z 1200.849,A -85,B 0,C 180,E1 5866.694,E2 5866.694} C_VEL
LIN {X 0,Y 500.637,Z 1177.759,A -85,B 0,C 180,E1 5870.204,E2 5870.204} C_VEL
LIN {X 0,Y 503.18,Z 1147.625,A -85,B 0,C 180,E1 5873.635,E2 5873.635} C_VEL
LIN {X 0,Y 505.705,Z 1116.255,A -85,B 0,C 180,E1 5876.218,E2 5876.218} C_VEL
LIN {X 0,Y 507.949,Z 1082.317,A -85,B 0,C 180,E1 5878.197,E2 5878.197} C_VEL
LIN {X 0,Y 509.7,Z 1045.429,A -85,B 0,C 180,E1 5879.576,E2 5879.576} C_VEL
LIN {X 0,Y 509.913,Z 1020.429,A -85,B 0,C 180,E1 5880.138,E2 5880.138} C_VEL
LIN {X 0,Y 496.585,Z 989.03,A -85,B 0,C 180,E1 5881.632,E2 5881.632} C_VEL
LIN {X 0,Y 496.249,Z 989.03,A -85,B 0,C 180,E1 5887.761,E2 5887.761} C_VEL
LIN {X 0,Y 496.302,Z 989.03,A -85,B 0,C 180,E1 5894.369,E2 5894.369} C_VEL
LIN {X 0,Y 496.382,Z 989.03,A -85,B 0,C 180,E1 5900.33,E2 5900.33} C_VEL
LIN {X 0,Y 496.375,Z 989.03,A -85,B 0,C 180,E1 5906.826,E2 5906.826} C_VEL
LIN {X 0,Y 496.468,Z 989.03,A -85,B 0,C 180,E1 5912.877,E2 5912.877} C_VEL
LIN {X 0,Y 496.663,Z 989.03,A -85,B 0,C 180,E1 5918.619,E2 5918.619} C_VEL
LIN {X 0,Y 496.853,Z 989.03,A -85,B 0,C 180,E1 5924.138,E2 5924.138} C_VEL
LIN {X 0,Y 496.868,Z 989.03,A -85,B 0,C 180,E1 5929.502,E2 5929.502} C_VEL
LIN {X 0,Y 496.998,Z 989.03,A -85,B 0,C 180,E1 5934.774,E2 5934.774} C_VEL
LIN {X 0,Y 497.219,Z 989.03,A -85,B 0,C 180,E1 5941.739,E2 5941.739} C_VEL
LIN {X 0,Y 496.98,Z 989.03,A -85,B 0,C 180,E1 5946.976,E2 5946.976} C_VEL
LIN {X 0,Y 496.784,Z 989.03,A -85,B 0,C 180,E1 5952.276,E2 5952.276} C_VEL
LIN {X 0,Y 496.694,Z 989.03,A -85,B 0,C 180,E1 5957.686,E2 5957.686} C_VEL
LIN {X 0,Y 496.536,Z 989.03,A -85,B 0,C 180,E1 5963.27,E2 5963.27} C_VEL
LIN {X 0,Y 496.448,Z 989.03,A -85,B 0,C 180,E1 5969.099,E2 5969.099} C_VEL
LIN {X 0,Y 496.395,Z 989.03,A -85,B 0,C 180,E1 5975.28,E2 5975.28} C_VEL
LIN {X 0,Y 496.347,Z 989.03,A -85,B 0,C 180,E1 5980.534,E2 5980.534} C_VEL
LIN {X 0,Y 496.293,Z 989.03,A -85,B 0,C 180,E1 5985.724,E2 5985.724} C_VEL
LIN {X 0,Y 492.27,Z 989.03,A -85,B 0,C 180,E1 5987.698,E2 5987.698} C_VEL
LIN {X 0,Y 488.328,Z 989.03,A -85,B 0,C 180,E1 5989.703,E2 5989.703} C_VEL
LIN {X 0,Y 488.385,Z 989.587,A -85,B 0,C 180,E1 5990.433,E2 5990.433} C_VEL
LIN {X 0,Y 497.979,Z 1016.451,A -85,B 0,C 180,E1 5992.971,E2 5992.971} C_VEL
LIN {X 0,Y 506.119,Z 1028.129,A -85,B 0,C 180,E1 5994.146,E2 5994.146} C_VEL
LIN {X 0,Y 507.803,Z 1030.598,A -85,B 0,C 180,E1 5994.302,E2 5994.302} C_VEL
LIN {X 0,Y 506.741,Z 1082.657,A -85,B 0,C 180,E1 5995.274,E2 5995.274} C_VEL
LIN {X 0,Y 504.693,Z 1122.469,A -85,B 0,C 180,E1 5996.677,E2 5996.677} C_VEL
LIN {X 0,Y 501.918,Z 1157.655,A -85,B 0,C 180,E1 5998.6,E2 5998.6} C_VEL
LIN {X 0,Y 498.597,Z 1193.44,A -85,B 0,C 180,E1 6001.361,E2 6001.361} C_VEL
LIN {X 0,Y 495.522,Z 1224.889,A -85,B 0,C 180,E1 6004.637,E2 6004.637} C_VEL
LIN {X 0,Y 492.912,Z 1252.784,A -85,B 0,C 180,E1 6008.449,E2 6008.449} C_VEL
LIN {X 0,Y 490.971,Z 1275.865,A -85,B 0,C 180,E1 6012.678,E2 6012.678} C_VEL
LIN {X 0,Y 489.924,Z 1293.574,A -85,B 0,C 180,E1 6017.1,E2 6017.1} C_VEL
LIN {X 0,Y 489.505,Z 1304.67,A -85,B 0,C 180,E1 6021.136,E2 6021.136} C_VEL
LIN {X 0,Y 489.294,Z 1310.996,A -85,B 0,C 180,E1 6024.695,E2 6024.695} C_VEL
LIN {X 0,Y 489.311,Z 1314.113,A -85,B 0,C 180,E1 6028.236,E2 6028.236} C_VEL
LIN {X 0,Y 489.386,Z 1314.111,A -85,B 0,C 180,E1 6031.77,E2 6031.77} C_VEL
LIN {X 0,Y 489.435,Z 1309.699,A -85,B 0,C 180,E1 6036.199,E2 6036.199} C_VEL
LIN {X 0,Y 489.577,Z 1300.258,A -85,B 0,C 180,E1 6040.661,E2 6040.661} C_VEL
LIN {X 0,Y 490.268,Z 1287.059,A -85,B 0,C 180,E1 6044.714,E2 6044.714} C_VEL
LIN {X 0,Y 491.633,Z 1267.288,A -85,B 0,C 180,E1 6049.038,E2 6049.038} C_VEL
LIN {X 0,Y 493.877,Z 1241.938,A -85,B 0,C 180,E1 6053.17,E2 6053.17} C_VEL
LIN {X 0,Y 496.819,Z 1211.418,A -85,B 0,C 180,E1 6056.879,E2 6056.879} C_VEL
LIN {X 0,Y 500.006,Z 1178.865,A -85,B 0,C 180,E1 6059.87,E2 6059.87} C_VEL
LIN {X 0,Y 503.303,Z 1141.972,A -85,B 0,C 180,E1 6062.348,E2 6062.348} C_VEL
LIN {X 0,Y 505.493,Z 1107.383,A -85,B 0,C 180,E1 6063.926,E2 6063.926} C_VEL
LIN {X 0,Y 507.089,Z 1066.206,A -85,B 0,C 180,E1 6065.026,E2 6065.026} C_VEL
LIN {X 0,Y 506.826,Z 1028.941,A -85,B 0,C 180,E1 6065.627,E2 6065.627} C_VEL
LIN {X 0,Y 498.751,Z 1018.445,A -85,B 0,C 180,E1 6066.336,E2 6066.336} C_VEL
LIN {X 0,Y 491.677,Z 1003.443,A -85,B 0,C 180,E1 6067.472,E2 6067.472} C_VEL
LIN {X 0,Y 488.598,Z 989.03,A -85,B 0,C 180,E1 6068.459,E2 6068.459} C_VEL
LIN {X 0,Y 488.418,Z 989.03,A -85,B 0,C 180,E1 6075.291,E2 6075.291} C_VEL
LIN {X 0,Y 488.318,Z 989.03,A -85,B 0,C 180,E1 6081.828,E2 6081.828} C_VEL
LIN {X 0,Y 488.554,Z 989.03,A -85,B 0,C 180,E1 6088.327,E2 6088.327} C_VEL
LIN {X 0,Y 488.56,Z 989.03,A -85,B 0,C 180,E1 6094.38,E2 6094.38} C_VEL
LIN {X 0,Y 488.734,Z 989.03,A -85,B 0,C 180,E1 6097.187,E2 6097.187} C_VEL
LIN {X 0,Y 496.245,Z 1016.282,A -85,B 0,C 180,E1 6098.032,E2 6098.032} C_VEL
LIN {X 0,Y 495.648,Z 1047.569,A -85,B 0,C 180,E1 6098.913,E2 6098.913} C_VEL
LIN {X 0,Y 494.42,Z 1076.804,A -85,B 0,C 180,E1 6100.463,E2 6100.463} C_VEL
LIN {X 0,Y 492.93,Z 1102.996,A -85,B 0,C 180,E1 6102.634,E2 6102.634} C_VEL
LIN {X 0,Y 491.528,Z 1125.909,A -85,B 0,C 180,E1 6105.446,E2 6105.446} C_VEL
LIN {X 0,Y 490.317,Z 1143.824,A -85,B 0,C 180,E1 6108.685,E2 6108.685} C_VEL
LIN {X 0,Y 489.789,Z 1155.872,A -85,B 0,C 180,E1 6112.031,E2 6112.031} C_VEL
LIN {X 0,Y 489.528,Z 1162.981,A -85,B 0,C 180,E1 6115.58,E2 6115.58} C_VEL
LIN {X 0,Y 489.476,Z 1165.108,A -85,B 0,C 180,E1 6118.233,E2 6118.233} C_VEL
LIN {X 0,Y 489.558,Z 1163.557,A -85,B 0,C 180,E1 6121.766,E2 6121.766} C_VEL
LIN {X 0,Y 489.786,Z 1155.958,A -85,B 0,C 180,E1 6125.746,E2 6125.746} C_VEL
LIN {X 0,Y 490.272,Z 1142.954,A -85,B 0,C 180,E1 6129.283,E2 6129.283} C_VEL
LIN {X 0,Y 491.271,Z 1125.345,A -85,B 0,C 180,E1 6132.415,E2 6132.415} C_VEL
LIN {X 0,Y 492.615,Z 1103.557,A -85,B 0,C 180,E1 6135.077,E2 6135.077} C_VEL
LIN {X 0,Y 494.174,Z 1076.942,A -85,B 0,C 180,E1 6137.32,E2 6137.32} C_VEL
LIN {X 0,Y 495.44,Z 1048.555,A -85,B 0,C 180,E1 6138.885,E2 6138.885} C_VEL
LIN {X 0,Y 496.099,Z 1016.797,A -85,B 0,C 180,E1 6139.865,E2 6139.865} C_VEL
LIN {X 0,Y 493.835,Z 1005.025,A -85,B 0,C 180,E1 6140.181,E2 6140.181} C_VEL
LIN {X 0,Y 488.864,Z 989.03,A -85,B 0,C 180,E1 6140.7,E2 6140.7} C_VEL
LIN {X 0,Y 488.507,Z 989.03,A -85,B 0,C 180,E1 6146.376,E2 6146.376} C_VEL
LIN {X 0,Y 488.469,Z 989.03,A -85,B 0,C 180,E1 6151.678,E2 6151.678} C_VEL
LIN {X 0,Y 488.297,Z 989.03,A -85,B 0,C 180,E1 6158.173,E2 6158.173} C_VEL
LIN {X 0,Y 488.428,Z 989.03,A -85,B 0,C 180,E1 6164.711,E2 6164.711} C_VEL
LIN {X 0,Y 488.455,Z 989.03,A -85,B 0,C 180,E1 6170.56,E2 6170.56} C_VEL
LIN {X 0,Y 488.443,Z 989.03,A -85,B 0,C 180,E1 6176.522,E2 6176.522} C_VEL
LIN {X 0,Y 488.488,Z 989.03,A -85,B 0,C 180,E1 6177.721,E2 6177.721} C_VEL
LIN {X 0,Y 503.492,Z 1025.491,A -85,B 0,C 180,E1 6179.434,E2 6179.434} C_VEL
LIN {X 0,Y 502.236,Z 1060.684,A -85,B 0,C 180,E1 6180.364,E2 6180.364} C_VEL
LIN {X 0,Y 500.274,Z 1094.296,A -85,B 0,C 180,E1 6181.876,E2 6181.876} C_VEL
LIN {X 0,Y 497.717,Z 1127.509,A -85,B 0,C 180,E1 6184.085,E2 6184.085} C_VEL
LIN {X 0,Y 494.926,Z 1158.716,A -85,B 0,C 180,E1 6187.001,E2 6187.001} C_VEL
LIN {X 0,Y 492.635,Z 1184.585,A -85,B 0,C 180,E1 6190.305,E2 6190.305} C_VEL
LIN {X 0,Y 490.784,Z 1208.42,A -85,B 0,C 180,E1 6194.389,E2 6194.389} C_VEL
LIN {X 0,Y 489.849,Z 1225.25,A -85,B 0,C 180,E1 6198.445,E2 6198.445} C_VEL
LIN {X 0,Y 489.538,Z 1235.495,A -85,B 0,C 180,E1 6202.023,E2 6202.023} C_VEL
LIN {X 0,Y 489.422,Z 1242.717,A -85,B 0,C 180,E1 6206.461,E2 6206.461} C_VEL
LIN {X 0,Y 489.327,Z 1244.498,A -85,B 0,C 180,E1 6209.997,E2 6209.997} C_VEL
LIN {X 0,Y 489.433,Z 1241.631,A -85,B 0,C 180,E1 6214.417,E2 6214.417} C_VEL
LIN {X 0,Y 489.607,Z 1233.081,A -85,B 0,C 180,E1 6218.862,E2 6218.862} C_VEL
LIN {X 0,Y 490.167,Z 1220.002,A -85,B 0,C 180,E1 6222.894,E2 6222.894} C_VEL
LIN {X 0,Y 491.266,Z 1200.851,A -85,B 0,C 180,E1 6226.963,E2 6226.963} C_VEL
LIN {X 0,Y 493.313,Z 1176.08,A -85,B 0,C 180,E1 6230.806,E2 6230.806} C_VEL
LIN {X 0,Y 495.977,Z 1147.627,A -85,B 0,C 180,E1 6234.059,E2 6234.059} C_VEL
LIN {X 0,Y 498.683,Z 1115.674,A -85,B 0,C 180,E1 6236.703,E2 6236.703} C_VEL
LIN {X 0,Y 501.115,Z 1081.71,A -85,B 0,C 180,E1 6238.678,E2 6238.678} C_VEL
LIN {X 0,Y 502.9,Z 1045.547,A -85,B 0,C 180,E1 6240.028,E2 6240.028} C_VEL
LIN {X 0,Y 502.957,Z 1022.347,A -85,B 0,C 180,E1 6240.574,E2 6240.574} C_VEL
LIN {X 0,Y 488.593,Z 989.03,A -85,B 0,C 180,E1 6242.224,E2 6242.224} C_VEL
LIN {X 0,Y 488.323,Z 989.03,A -85,B 0,C 180,E1 6248.17,E2 6248.17} C_VEL
LIN {X 0,Y 488.392,Z 989.03,A -85,B 0,C 180,E1 6254.716,E2 6254.716} C_VEL
LIN {X 0,Y 488.457,Z 989.03,A -85,B 0,C 180,E1 6260.561,E2 6260.561} C_VEL
LIN {X 0,Y 488.451,Z 989.03,A -85,B 0,C 180,E1 6266.522,E2 6266.522} C_VEL
LIN {X 0,Y 488.54,Z 989.03,A -85,B 0,C 180,E1 6272.4,E2 6272.4} C_VEL
LIN {X 0,Y 488.704,Z 989.03,A -85,B 0,C 180,E1 6278.253,E2 6278.253} C_VEL
LIN {X 0,Y 488.91,Z 989.03,A -85,B 0,C 180,E1 6283.873,E2 6283.873} C_VEL
LIN {X 0,Y 488.976,Z 989.03,A -85,B 0,C 180,E1 6289.33,E2 6289.33} C_VEL
LIN {X 0,Y 489.084,Z 989.03,A -85,B 0,C 180,E1 6294.69,E2 6294.69} C_VEL
LIN {X 0,Y 489.218,Z 989.03,A -85,B 0,C 180,E1 6300,E2 6300} C_VEL
LIN {X 0,Y 489.107,Z 989.03,A -85,B 0,C 180,E1 6305.311,E2 6305.311} C_VEL
LIN {X 0,Y 488.923,Z 989.03,A -85,B 0,C 180,E1 6310.672,E2 6310.672} C_VEL
LIN {X 0,Y 488.741,Z 989.03,A -85,B 0,C 180,E1 6316.842,E2 6316.842} C_VEL
LIN {X 0,Y 488.661,Z 989.03,A -85,B 0,C 180,E1 6322.122,E2 6322.122} C_VEL
LIN {X 0,Y 488.543,Z 989.03,A -85,B 0,C 180,E1 6327.6,E2 6327.6} C_VEL
LIN {X 0,Y 488.43,Z 989.03,A -85,B 0,C 180,E1 6333.786,E2 6333.786} C_VEL
LIN {X 0,Y 488.447,Z 989.03,A -85,B 0,C 180,E1 6340.447,E2 6340.447} C_VEL
LIN {X 0,Y 488.336,Z 989.03,A -85,B 0,C 180,E1 6345.713,E2 6345.713} C_VEL
LIN {X 0,Y 488.328,Z 989.03,A -85,B 0,C 180,E1 6349.703,E2 6349.703} C_VEL
LIN {X 0,Y 489.049,Z 992.368,A -85,B 0,C 180,E1 6350.578,E2 6350.578} C_VEL
LIN {X 0,Y 489.642,Z 999.28,A -85,B 0,C 180,E1 6351.208,E2 6351.208} C_VEL
LIN {X 0,Y 488.808,Z 1015.109,A -85,B 0,C 180,E1 6352.249,E2 6352.249} C_VEL
LIN {X 0,Y 489.107,Z 1016.019,A -85,B 0,C 180,E1 6352.333,E2 6352.333} C_VEL
LIN {X 0,Y 495.778,Z 1027.473,A -85,B 0,C 180,E1 6353.393,E2 6353.393} C_VEL
LIN {X 0,Y 500.889,Z 1033.596,A -85,B 0,C 180,E1 6353.868,E2 6353.868} C_VEL
LIN {X 0,Y 499.862,Z 1082.5,A -85,B 0,C 180,E1 6354.824,E2 6354.824} C_VEL
LIN {X 0,Y 497.606,Z 1122.601,A -85,B 0,C 180,E1 6356.275,E2 6356.275} C_VEL
LIN {X 0,Y 494.659,Z 1161.157,A -85,B 0,C 180,E1 6358.38,E2 6358.38} C_VEL
LIN {X 0,Y 491.415,Z 1194.351,A -85,B 0,C 180,E1 6360.992,E2 6360.992} C_VEL
LIN {X 0,Y 488.062,Z 1225.932,A -85,B 0,C 180,E1 6364.354,E2 6364.354} C_VEL
LIN {X 0,Y 485.333,Z 1252.788,A -85,B 0,C 180,E1 6368.096,E2 6368.096} C_VEL
LIN {X 0,Y 483.213,Z 1276.394,A -85,B 0,C 180,E1 6372.506,E2 6372.506} C_VEL
LIN {X 0,Y 482.066,Z 1293.86,A -85,B 0,C 180,E1 6376.98,E2 6376.98} C_VEL
LIN {X 0,Y 481.646,Z 1304.668,A -85,B 0,C 180,E1 6380.991,E2 6380.991} C_VEL
LIN {X 0,Y 481.404,Z 1310.992,A -85,B 0,C 180,E1 6384.607,E2 6384.607} C_VEL
LIN {X 0,Y 481.423,Z 1314.113,A -85,B 0,C 180,E1 6388.207,E2 6388.207} C_VEL
LIN {X 0,Y 481.485,Z 1314.111,A -85,B 0,C 180,E1 6391.8,E2 6391.8} C_VEL
LIN {X 0,Y 481.55,Z 1309.696,A -85,B 0,C 180,E1 6396.3,E2 6396.3} C_VEL
LIN {X 0,Y 481.714,Z 1300.256,A -85,B 0,C 180,E1 6400.837,E2 6400.837} C_VEL
LIN {X 0,Y 482.616,Z 1285.266,A -85,B 0,C 180,E1 6405.417,E2 6405.417} C_VEL
LIN {X 0,Y 484.292,Z 1263.612,A -85,B 0,C 180,E1 6410.049,E2 6410.049} C_VEL
LIN {X 0,Y 486.704,Z 1238.479,A -85,B 0,C 180,E1 6414.021,E2 6414.021} C_VEL
LIN {X 0,Y 489.978,Z 1207.823,A -85,B 0,C 180,E1 6417.699,E2 6417.699} C_VEL
LIN {X 0,Y 493.602,Z 1173.157,A -85,B 0,C 180,E1 6420.784,E2 6420.784} C_VEL
LIN {X 0,Y 496.175,Z 1140.404,A -85,B 0,C 180,E1 6422.807,E2 6422.807} C_VEL
LIN {X 0,Y 498.357,Z 1098.482,A -85,B 0,C 180,E1 6424.532,E2 6424.532} C_VEL
LIN {X 0,Y 499.977,Z 1054.036,A -85,B 0,C 180,E1 6425.58,E2 6425.58} C_VEL
LIN {X 0,Y 499.497,Z 1032.437,A -85,B 0,C 180,E1 6425.935,E2 6425.935} C_VEL
LIN {X 0,Y 488.123,Z 1015.839,A -85,B 0,C 180,E1 6426.898,E2 6426.898} C_VEL
LIN {X 0,Y 482.067,Z 995.839,A -85,B 0,C 180,E1 6428.334,E2 6428.334} C_VEL
LIN {X 0,Y 480.624,Z 989.03,A -85,B 0,C 180,E1 6428.904,E2 6428.904} C_VEL
LIN {X 0,Y 480.474,Z 989.03,A -85,B 0,C 180,E1 6433.753,E2 6433.753} C_VEL
LIN {X 0,Y 480.417,Z 989.03,A -85,B 0,C 180,E1 6438.932,E2 6438.932} C_VEL
LIN {X 0,Y 480.503,Z 989.03,A -85,B 0,C 180,E1 6445.579,E2 6445.579} C_VEL
LIN {X 0,Y 480.595,Z 989.03,A -85,B 0,C 180,E1 6451.903,E2 6451.903} C_VEL
LIN {X 0,Y 480.804,Z 989.452,A -85,B 0,C 180,E1 6456.771,E2 6456.771} C_VEL
LIN {X 0,Y 488.898,Z 1016.934,A -85,B 0,C 180,E1 6457.702,E2 6457.702} C_VEL
LIN {X 0,Y 488.351,Z 1048.535,A -85,B 0,C 180,E1 6458.585,E2 6458.585} C_VEL
LIN {X 0,Y 487.165,Z 1076.856,A -85,B 0,C 180,E1 6460.079,E2 6460.079} C_VEL
LIN {X 0,Y 485.631,Z 1103.235,A -85,B 0,C 180,E1 6462.248,E2 6462.248} C_VEL
LIN {X 0,Y 484.171,Z 1124.968,A -85,B 0,C 180,E1 6464.867,E2 6464.867} C_VEL
LIN {X 0,Y 482.82,Z 1143.219,A -85,B 0,C 180,E1 6468.05,E2 6468.05} C_VEL
LIN {X 0,Y 482.163,Z 1155.962,A -85,B 0,C 180,E1 6471.451,E2 6471.451} C_VEL
LIN {X 0,Y 481.842,Z 1163.135,A -85,B 0,C 180,E1 6474.609,E2 6474.609} C_VEL
LIN {X 0,Y 481.702,Z 1166.477,A -85,B 0,C 180,E1 6478.205,E2 6478.205} C_VEL
LIN {X 0,Y 481.794,Z 1164.903,A -85,B 0,C 180,E1 6481.794,E2 6481.794} C_VEL
LIN {X 0,Y 481.977,Z 1158.357,A -85,B 0,C 180,E1 6485.389,E2 6485.389} C_VEL
LIN {X 0,Y 482.521,Z 1146.17,A -85,B 0,C 180,E1 6488.995,E2 6488.995} C_VEL
LIN {X 0,Y 483.543,Z 1128.001,A -85,B 0,C 180,E1 6492.388,E2 6492.388} C_VEL
LIN {X 0,Y 485.003,Z 1106.133,A -85,B 0,C 180,E1 6495.173,E2 6495.173} C_VEL
LIN {X 0,Y 486.66,Z 1079.718,A -85,B 0,C 180,E1 6497.479,E2 6497.479} C_VEL
LIN {X 0,Y 488.006,Z 1051.11,A -85,B 0,C 180,E1 6499.126,E2 6499.126} C_VEL
LIN {X 0,Y 488.831,Z 1020.325,A -85,B 0,C 180,E1 6500.136,E2 6500.136} C_VEL
LIN {X 0,Y 487.089,Z 1008.556,A -85,B 0,C 180,E1 6500.441,E2 6500.441} C_VEL
LIN {X 0,Y 480.896,Z 989.03,A -85,B 0,C 180,E1 6501.17,E2 6501.17} C_VEL
LIN {X 0,Y 480.647,Z 989.03,A -85,B 0,C 180,E1 6506.073,E2 6506.073} C_VEL
LIN {X 0,Y 480.535,Z 989.03,A -85,B 0,C 180,E1 6512.264,E2 6512.264} C_VEL
LIN {X 0,Y 480.36,Z 989.03,A -85,B 0,C 180,E1 6518.921,E2 6518.921} C_VEL
LIN {X 0,Y 480.445,Z 989.03,A -85,B 0,C 180,E1 6523.74,E2 6523.74} C_VEL
LIN {X 0,Y 480.485,Z 989.03,A -85,B 0,C 180,E1 6528.912,E2 6528.912} C_VEL
LIN {X 0,Y 480.492,Z 989.03,A -85,B 0,C 180,E1 6534.736,E2 6534.736} C_VEL
LIN {X 0,Y 480.575,Z 989.152,A -85,B 0,C 180,E1 6537.142,E2 6537.142} C_VEL
LIN {X 0,Y 496.461,Z 1026.258,A -85,B 0,C 180,E1 6538.963,E2 6538.963} C_VEL
LIN {X 0,Y 495.304,Z 1063.417,A -85,B 0,C 180,E1 6539.997,E2 6539.997} C_VEL
LIN {X 0,Y 493.144,Z 1097.913,A -85,B 0,C 180,E1 6541.619,E2 6541.619} C_VEL
LIN {X 0,Y 490.255,Z 1131.641,A -85,B 0,C 180,E1 6543.967,E2 6543.967} C_VEL
LIN {X 0,Y 487.421,Z 1161.321,A -85,B 0,C 180,E1 6546.867,E2 6546.867} C_VEL
LIN {X 0,Y 484.983,Z 1186.717,A -85,B 0,C 180,E1 6550.218,E2 6550.218} C_VEL
LIN {X 0,Y 483.052,Z 1208.585,A -85,B 0,C 180,E1 6554.133,E2 6554.133} C_VEL
LIN {X 0,Y 482.005,Z 1225.246,A -85,B 0,C 180,E1 6558.255,E2 6558.255} C_VEL
LIN {X 0,Y 481.657,Z 1235.493,A -85,B 0,C 180,E1 6561.892,E2 6561.892} C_VEL
LIN {X 0,Y 481.543,Z 1242.716,A -85,B 0,C 180,E1 6566.403,E2 6566.403} C_VEL
LIN {X 0,Y 481.434,Z 1244.498,A -85,B 0,C 180,E1 6569.997,E2 6569.997} C_VEL
LIN {X 0,Y 481.554,Z 1241.632,A -85,B 0,C 180,E1 6574.49,E2 6574.49} C_VEL
LIN {X 0,Y 481.735,Z 1233.082,A -85,B 0,C 180,E1 6579.008,E2 6579.008} C_VEL
LIN {X 0,Y 482.404,Z 1218.695,A -85,B 0,C 180,E1 6583.45,E2 6583.45} C_VEL
LIN {X 0,Y 483.804,Z 1199.053,A -85,B 0,C 180,E1 6587.637,E2 6587.637} C_VEL
LIN {X 0,Y 486.042,Z 1175.123,A -85,B 0,C 180,E1 6591.353,E2 6591.353} C_VEL
LIN {X 0,Y 488.933,Z 1146.073,A -85,B 0,C 180,E1 6594.642,E2 6594.642} C_VEL
LIN {X 0,Y 491.777,Z 1114.345,A -85,B 0,C 180,E1 6597.252,E2 6597.252} C_VEL
LIN {X 0,Y 494.395,Z 1079.931,A -85,B 0,C 180,E1 6599.23,E2 6599.23} C_VEL
LIN {X 0,Y 496.226,Z 1043.284,A -85,B 0,C 180,E1 6600.55,E2 6600.55} C_VEL
LIN {X 0,Y 496.194,Z 1024.723,A -85,B 0,C 180,E1 6600.999,E2 6600.999} C_VEL
LIN {X 0,Y 480.65,Z 989.03,A -85,B 0,C 180,E1 6602.794,E2 6602.794} C_VEL
LIN {X 0,Y 480.394,Z 989.03,A -85,B 0,C 180,E1 6608.917,E2 6608.917} C_VEL
LIN {X 0,Y 480.402,Z 989.03,A -85,B 0,C 180,E1 6613.745,E2 6613.745} C_VEL
LIN {X 0,Y 480.484,Z 989.03,A -85,B 0,C 180,E1 6618.912,E2 6618.912} C_VEL
LIN {X 0,Y 480.494,Z 989.03,A -85,B 0,C 180,E1 6624.736,E2 6624.736} C_VEL
LIN {X 0,Y 480.534,Z 989.03,A -85,B 0,C 180,E1 6629.84,E2 6629.84} C_VEL
LIN {X 0,Y 480.71,Z 989.03,A -85,B 0,C 180,E1 6635.917,E2 6635.917} C_VEL
LIN {X 0,Y 480.894,Z 989.03,A -85,B 0,C 180,E1 6641.713,E2 6641.713} C_VEL
LIN {X 0,Y 481.041,Z 989.03,A -85,B 0,C 180,E1 6647.316,E2 6647.316} C_VEL
LIN {X 0,Y 481.093,Z 989.03,A -85,B 0,C 180,E1 6652.793,E2 6652.793} C_VEL
LIN {X 0,Y 481.201,Z 989.03,A -85,B 0,C 180,E1 6658.203,E2 6658.203} C_VEL
LIN {X 0,Y 481.193,Z 989.03,A -85,B 0,C 180,E1 6663.596,E2 6663.596} C_VEL
LIN {X 0,Y 481.02,Z 989.03,A -85,B 0,C 180,E1 6669.024,E2 6669.024} C_VEL
LIN {X 0,Y 480.911,Z 989.03,A -85,B 0,C 180,E1 6674.538,E2 6674.538} C_VEL
LIN {X 0,Y 480.802,Z 989.03,A -85,B 0,C 180,E1 6680.196,E2 6680.196} C_VEL
LIN {X 0,Y 480.661,Z 989.03,A -85,B 0,C 180,E1 6686.072,E2 6686.072} C_VEL
LIN {X 0,Y 480.492,Z 989.03,A -85,B 0,C 180,E1 6692.268,E2 6692.268} C_VEL
LIN {X 0,Y 480.561,Z 989.03,A -85,B 0,C 180,E1 6698.902,E2 6698.902} C_VEL
LIN {X 0,Y 480.458,Z 989.03,A -85,B 0,C 180,E1 6703.752,E2 6703.752} C_VEL
LIN {X 0,Y 480.428,Z 989.075,A -85,B 0,C 180,E1 6709.783,E2 6709.783} C_VEL
LIN {X 0,Y 489.107,Z 1016.019,A -85,B 0,C 180,E1 6712.333,E2 6712.333} C_VEL
LIN {X 0,Y 492.948,Z 1035.553,A -85,B 0,C 180,E1 6713.324,E2 6713.324} C_VEL
LIN {X 0,Y 494.08,Z 1037.167,A -85,B 0,C 180,E1 6713.437,E2 6713.437} C_VEL
LIN {X 0,Y 492.973,Z 1082.765,A -85,B 0,C 180,E1 6714.377,E2 6714.377} C_VEL
LIN {X 0,Y 490.531,Z 1122.49,A -85,B 0,C 180,E1 6715.85,E2 6715.85} C_VEL
LIN {X 0,Y 487.241,Z 1162.565,A -85,B 0,C 180,E1 6718.103,E2 6718.103} C_VEL
LIN {X 0,Y 483.905,Z 1198.188,A -85,B 0,C 180,E1 6720.897,E2 6720.897} C_VEL
LIN {X 0,Y 480.331,Z 1229.792,A -85,B 0,C 180,E1 6724.41,E2 6724.41} C_VEL
LIN {X 0,Y 477.283,Z 1257.025,A -85,B 0,C 180,E1 6728.453,E2 6728.453} C_VEL
LIN {X 0,Y 475.283,Z 1279.004,A -85,B 0,C 180,E1 6732.785,E2 6732.785} C_VEL
LIN {X 0,Y 474.153,Z 1294.976,A -85,B 0,C 180,E1 6737.131,E2 6737.131} C_VEL
LIN {X 0,Y 473.675,Z 1306.603,A -85,B 0,C 180,E1 6741.776,E2 6741.776} C_VEL
LIN {X 0,Y 473.501,Z 1312.942,A -85,B 0,C 180,E1 6746.349,E2 6746.349} C_VEL
LIN {X 0,Y 473.538,Z 1314.5,A -85,B 0,C 180,E1 6750.004,E2 6750.004} C_VEL
LIN {X 0,Y 473.479,Z 1312.944,A -85,B 0,C 180,E1 6753.658,E2 6753.658} C_VEL
LIN {X 0,Y 473.7,Z 1306.579,A -85,B 0,C 180,E1 6758.232,E2 6758.232} C_VEL
LIN {X 0,Y 474.227,Z 1294.96,A -85,B 0,C 180,E1 6762.874,E2 6762.874} C_VEL
LIN {X 0,Y 475.437,Z 1277.945,A -85,B 0,C 180,E1 6767.446,E2 6767.446} C_VEL
LIN {X 0,Y 477.63,Z 1254.166,A -85,B 0,C 180,E1 6772.036,E2 6772.036} C_VEL
LIN {X 0,Y 480.486,Z 1227.796,A -85,B 0,C 180,E1 6775.838,E2 6775.838} C_VEL
LIN {X 0,Y 483.985,Z 1197.186,A -85,B 0,C 180,E1 6779.194,E2 6779.194} C_VEL
LIN {X 0,Y 486.672,Z 1166.538,A -85,B 0,C 180,E1 6781.544,E2 6781.544} C_VEL
LIN {X 0,Y 489.471,Z 1125.818,A -85,B 0,C 180,E1 6783.777,E2 6783.777} C_VEL
LIN {X 0,Y 491.732,Z 1082.702,A -85,B 0,C 180,E1 6785.317,E2 6785.317} C_VEL
LIN {X 0,Y 492.486,Z 1036.037,A -85,B 0,C 180,E1 6786.235,E2 6786.235} C_VEL
LIN {X 0,Y 479.258,Z 1015.279,A -85,B 0,C 180,E1 6787.299,E2 6787.299} C_VEL
LIN {X 0,Y 472.658,Z 989.03,A -85,B 0,C 180,E1 6789.256,E2 6789.256} C_VEL
LIN {X 0,Y 472.461,Z 989.03,A -85,B 0,C 180,E1 6795.361,E2 6795.361} C_VEL
LIN {X 0,Y 472.413,Z 989.03,A -85,B 0,C 180,E1 6800.296,E2 6800.296} C_VEL
LIN {X 0,Y 472.583,Z 989.03,A -85,B 0,C 180,E1 6806.129,E2 6806.129} C_VEL
LIN {X 0,Y 472.698,Z 989.03,A -85,B 0,C 180,E1 6811.391,E2 6811.391} C_VEL
LIN {X 0,Y 472.849,Z 989.067,A -85,B 0,C 180,E1 6816.301,E2 6816.301} C_VEL
LIN {X 0,Y 481.495,Z 1016.731,A -85,B 0,C 180,E1 6817.338,E2 6817.338} C_VEL
LIN {X 0,Y 481.05,Z 1048.245,A -85,B 0,C 180,E1 6818.198,E2 6818.198} C_VEL
LIN {X 0,Y 479.951,Z 1076.382,A -85,B 0,C 180,E1 6819.656,E2 6819.656} C_VEL
LIN {X 0,Y 478.283,Z 1103.357,A -85,B 0,C 180,E1 6821.847,E2 6821.847} C_VEL
LIN {X 0,Y 476.668,Z 1126.521,A -85,B 0,C 180,E1 6824.648,E2 6824.648} C_VEL
LIN {X 0,Y 475.216,Z 1144.645,A -85,B 0,C 180,E1 6827.856,E2 6827.856} C_VEL
LIN {X 0,Y 474.469,Z 1157.395,A -85,B 0,C 180,E1 6831.311,E2 6831.311} C_VEL
LIN {X 0,Y 474.115,Z 1164.529,A -85,B 0,C 180,E1 6834.521,E2 6834.521} C_VEL
LIN {X 0,Y 473.943,Z 1167.843,A -85,B 0,C 180,E1 6838.175,E2 6838.175} C_VEL
LIN {X 0,Y 474.035,Z 1166.248,A -85,B 0,C 180,E1 6841.824,E2 6841.824} C_VEL
LIN {X 0,Y 474.232,Z 1159.646,A -85,B 0,C 180,E1 6845.477,E2 6845.477} C_VEL
LIN {X 0,Y 474.832,Z 1147.389,A -85,B 0,C 180,E1 6849.142,E2 6849.142} C_VEL
LIN {X 0,Y 475.949,Z 1129.205,A -85,B 0,C 180,E1 6852.589,E2 6852.589} C_VEL
LIN {X 0,Y 477.47,Z 1107.294,A -85,B 0,C 180,E1 6855.419,E2 6855.419} C_VEL
LIN {X 0,Y 479.227,Z 1080.917,A -85,B 0,C 180,E1 6857.76,E2 6857.76} C_VEL
LIN {X 0,Y 480.664,Z 1051.745,A -85,B 0,C 180,E1 6859.457,E2 6859.457} C_VEL
LIN {X 0,Y 481.511,Z 1021.628,A -85,B 0,C 180,E1 6860.464,E2 6860.464} C_VEL
LIN {X 0,Y 479.793,Z 1010.203,A -85,B 0,C 180,E1 6860.769,E2 6860.769} C_VEL
LIN {X 0,Y 472.965,Z 989.03,A -85,B 0,C 180,E1 6861.525,E2 6861.525} C_VEL
LIN {X 0,Y 472.673,Z 989.03,A -85,B 0,C 180,E1 6866.621,E2 6866.621} C_VEL
LIN {X 0,Y 472.542,Z 989.03,A -85,B 0,C 180,E1 6872.877,E2 6872.877} C_VEL
LIN {X 0,Y 472.464,Z 989.03,A -85,B 0,C 180,E1 6877.359,E2 6877.359} C_VEL
LIN {X 0,Y 472.451,Z 989.03,A -85,B 0,C 180,E1 6882.718,E2 6882.718} C_VEL
LIN {X 0,Y 472.478,Z 989.03,A -85,B 0,C 180,E1 6887.872,E2 6887.872} C_VEL
LIN {X 0,Y 472.631,Z 989.03,A -85,B 0,C 180,E1 6892.954,E2 6892.954} C_VEL
LIN {X 0,Y 472.61,Z 989.03,A -85,B 0,C 180,E1 6896.493,E2 6896.493} C_VEL
LIN {X 0,Y 489.847,Z 1029.78,A -85,B 0,C 180,E1 6898.565,E2 6898.565} C_VEL
LIN {X 0,Y 488.41,Z 1065.469,A -85,B 0,C 180,E1 6899.593,E2 6899.593} C_VEL
LIN {X 0,Y 486.036,Z 1100.505,A -85,B 0,C 180,E1 6901.293,E2 6901.293} C_VEL
LIN {X 0,Y 482.944,Z 1134.057,A -85,B 0,C 180,E1 6903.715,E2 6903.715} C_VEL
LIN {X 0,Y 479.94,Z 1163.924,A -85,B 0,C 180,E1 6906.73,E2 6906.73} C_VEL
LIN {X 0,Y 477.161,Z 1190.303,A -85,B 0,C 180,E1 6910.362,E2 6910.362} C_VEL
LIN {X 0,Y 475.199,Z 1211.261,A -85,B 0,C 180,E1 6914.336,E2 6914.336} C_VEL
LIN {X 0,Y 474.123,Z 1226.934,A -85,B 0,C 180,E1 6918.522,E2 6918.522} C_VEL
LIN {X 0,Y 473.696,Z 1237.395,A -85,B 0,C 180,E1 6922.675,E2 6922.675} C_VEL
LIN {X 0,Y 473.638,Z 1242.715,A -85,B 0,C 180,E1 6926.343,E2 6926.343} C_VEL
LIN {X 0,Y 473.534,Z 1244.498,A -85,B 0,C 180,E1 6929.996,E2 6929.996} C_VEL
LIN {X 0,Y 473.669,Z 1241.632,A -85,B 0,C 180,E1 6934.565,E2 6934.565} C_VEL
LIN {X 0,Y 473.87,Z 1232.969,A -85,B 0,C 180,E1 6939.205,E2 6939.205} C_VEL
LIN {X 0,Y 474.641,Z 1219.49,A -85,B 0,C 180,E1 6943.583,E2 6943.583} C_VEL
LIN {X 0,Y 476.038,Z 1201.27,A -85,B 0,C 180,E1 6947.633,E2 6947.633} C_VEL
LIN {X 0,Y 478.343,Z 1178.36,A -85,B 0,C 180,E1 6951.333,E2 6951.333} C_VEL
LIN {X 0,Y 481.262,Z 1151.072,A -85,B 0,C 180,E1 6954.598,E2 6954.598} C_VEL
LIN {X 0,Y 484.461,Z 1118.559,A -85,B 0,C 180,E1 6957.419,E2 6957.419} C_VEL
LIN {X 0,Y 487.129,Z 1085.146,A -85,B 0,C 180,E1 6959.454,E2 6959.454} C_VEL
LIN {X 0,Y 489.169,Z 1049.123,A -85,B 0,C 180,E1 6960.875,E2 6960.875} C_VEL
LIN {X 0,Y 489.294,Z 1026.723,A -85,B 0,C 180,E1 6961.451,E2 6961.451} C_VEL
LIN {X 0,Y 472.693,Z 989.03,A -85,B 0,C 180,E1 6963.465,E2 6963.465} C_VEL
LIN {X 0,Y 472.41,Z 989.03,A -85,B 0,C 180,E1 6969.952,E2 6969.952} C_VEL
LIN {X 0,Y 472.454,Z 989.03,A -85,B 0,C 180,E1 6975.361,E2 6975.361} C_VEL
LIN {X 0,Y 472.552,Z 989.03,A -85,B 0,C 180,E1 6980.31,E2 6980.31} C_VEL
LIN {X 0,Y 472.538,Z 989.03,A -85,B 0,C 180,E1 6986.124,E2 6986.124} C_VEL
LIN {X 0,Y 472.652,Z 989.03,A -85,B 0,C 180,E1 6991.389,E2 6991.389} C_VEL
LIN {X 0,Y 472.871,Z 989.03,A -85,B 0,C 180,E1 6997.729,E2 6997.729} C_VEL
LIN {X 0,Y 473.036,Z 989.03,A -85,B 0,C 180,E1 7003.316,E2 7003.316} C_VEL
LIN {X 0,Y 473.146,Z 989.03,A -85,B 0,C 180,E1 7008.969,E2 7008.969} C_VEL
LIN {X 0,Y 473.253,Z 989.03,A -85,B 0,C 180,E1 7014.511,E2 7014.511} C_VEL
LIN {X 0,Y 473.439,Z 989.03,A -85,B 0,C 180,E1 7020,E2 7020} C_VEL
LIN {X 0,Y 473.279,Z 989.03,A -85,B 0,C 180,E1 7025.489,E2 7025.489} C_VEL
LIN {X 0,Y 473.093,Z 989.03,A -85,B 0,C 180,E1 7031.033,E2 7031.033} C_VEL
LIN {X 0,Y 472.913,Z 989.03,A -85,B 0,C 180,E1 7036.818,E2 7036.818} C_VEL
LIN {X 0,Y 472.81,Z 989.03,A -85,B 0,C 180,E1 7042.518,E2 7042.518} C_VEL
LIN {X 0,Y 472.652,Z 989.03,A -85,B 0,C 180,E1 7048.612,E2 7048.612} C_VEL
LIN {X 0,Y 472.588,Z 989.03,A -85,B 0,C 180,E1 7055.081,E2 7055.081} C_VEL
LIN {X 0,Y 472.548,Z 989.03,A -85,B 0,C 180,E1 7059.972,E2 7059.972} C_VEL
LIN {X 0,Y 472.445,Z 989.03,A -85,B 0,C 180,E1 7065.36,E2 7065.36} C_VEL
LIN {X 0,Y 472.535,Z 989.519,A -85,B 0,C 180,E1 7069.182,E2 7069.182} C_VEL
LIN {X 0,Y 484.779,Z 1024.36,A -85,B 0,C 180,E1 7072.497,E2 7072.497} C_VEL
LIN {X 0,Y 494.08,Z 1037.167,A -85,B 0,C 180,E1 7073.437,E2 7073.437} C_VEL
LIN {X 0,Y 495.663,Z 1043.536,A -85,B 0,C 180,E1 7073.657,E2 7073.657} C_VEL
LIN {X 0,Y 493.185,Z 1052.932,A -85,B 0,C 180,E1 7073.641,E2 7073.641} C_VEL
LIN {X 0,Y 486.962,Z 1069.061,A -85,B 0,C 180,E1 7073.557,E2 7073.557} C_VEL
LIN {X 0,Y 486.691,Z 1071.454,A -85,B 0,C 180,E1 7073.606,E2 7073.606} C_VEL
LIN {X 0,Y 484.126,Z 1113.02,A -85,B 0,C 180,E1 7074.993,E2 7074.993} C_VEL
LIN {X 0,Y 480.702,Z 1153.431,A -85,B 0,C 180,E1 7077.12,E2 7077.12} C_VEL
LIN {X 0,Y 477.11,Z 1191.326,A -85,B 0,C 180,E1 7079.963,E2 7079.963} C_VEL
LIN {X 0,Y 473.645,Z 1223.91,A -85,B 0,C 180,E1 7083.261,E2 7083.261} C_VEL
LIN {X 0,Y 470.403,Z 1251.595,A -85,B 0,C 180,E1 7087.16,E2 7087.16} C_VEL
LIN {X 0,Y 467.909,Z 1275.058,A -85,B 0,C 180,E1 7091.616,E2 7091.616} C_VEL
LIN {X 0,Y 466.607,Z 1292.046,A -85,B 0,C 180,E1 7095.968,E2 7095.968} C_VEL
LIN {X 0,Y 465.9,Z 1304.664,A -85,B 0,C 180,E1 7100.684,E2 7100.684} C_VEL
LIN {X 0,Y 465.63,Z 1310.984,A -85,B 0,C 180,E1 7104.424,E2 7104.424} C_VEL
LIN {X 0,Y 465.619,Z 1314.11,A -85,B 0,C 180,E1 7108.146,E2 7108.146} C_VEL
LIN {X 0,Y 465.672,Z 1314.11,A -85,B 0,C 180,E1 7111.861,E2 7111.861} C_VEL
LIN {X 0,Y 465.735,Z 1309.688,A -85,B 0,C 180,E1 7116.515,E2 7116.515} C_VEL
LIN {X 0,Y 466.023,Z 1300.25,A -85,B 0,C 180,E1 7121.207,E2 7121.207} C_VEL
LIN {X 0,Y 467.084,Z 1285.256,A -85,B 0,C 180,E1 7125.943,E2 7125.943} C_VEL
LIN {X 0,Y 469.058,Z 1263.605,A -85,B 0,C 180,E1 7130.729,E2 7130.729} C_VEL
LIN {X 0,Y 471.891,Z 1238.499,A -85,B 0,C 180,E1 7134.821,E2 7134.821} C_VEL
LIN {X 0,Y 474.777,Z 1213.4,A -85,B 0,C 180,E1 7137.906,E2 7137.906} C_VEL
LIN {X 0,Y 477.853,Z 1180.336,A -85,B 0,C 180,E1 7140.802,E2 7140.802} C_VEL
LIN {X 0,Y 481.003,Z 1140.876,A -85,B 0,C 180,E1 7143.315,E2 7143.315} C_VEL
LIN {X 0,Y 483.526,Z 1098.508,A -85,B 0,C 180,E1 7145.165,E2 7145.165} C_VEL
LIN {X 0,Y 485.46,Z 1054.821,A -85,B 0,C 180,E1 7146.288,E2 7146.288} C_VEL
LIN {X 0,Y 484.901,Z 1038.768,A -85,B 0,C 180,E1 7146.589,E2 7146.589} C_VEL
LIN {X 0,Y 471.969,Z 1017.13,A -85,B 0,C 180,E1 7147.705,E2 7147.705} C_VEL
LIN {X 0,Y 468.542,Z 1005.912,A -85,B 0,C 180,E1 7148.374,E2 7148.374} C_VEL
LIN {X 0,Y 464.709,Z 989.03,A -85,B 0,C 180,E1 7149.711,E2 7149.711} C_VEL
LIN {X 0,Y 464.532,Z 989.03,A -85,B 0,C 180,E1 7155.622,E2 7155.622} C_VEL
LIN {X 0,Y 464.491,Z 989.03,A -85,B 0,C 180,E1 7161.885,E2 7161.885} C_VEL
LIN {X 0,Y 464.664,Z 989.03,A -85,B 0,C 180,E1 7167.613,E2 7167.613} C_VEL
LIN {X 0,Y 464.779,Z 989.03,A -85,B 0,C 180,E1 7172.966,E2 7172.966} C_VEL
LIN {X 0,Y 464.911,Z 989.321,A -85,B 0,C 180,E1 7175.803,E2 7175.803} C_VEL
LIN {X 0,Y 474.281,Z 1018.509,A -85,B 0,C 180,E1 7176.996,E2 7176.996} C_VEL
LIN {X 0,Y 473.794,Z 1051.04,A -85,B 0,C 180,E1 7177.919,E2 7177.919} C_VEL
LIN {X 0,Y 472.484,Z 1080.412,A -85,B 0,C 180,E1 7179.512,E2 7179.512} C_VEL
LIN {X 0,Y 470.722,Z 1107.063,A -85,B 0,C 180,E1 7181.787,E2 7181.787} C_VEL
LIN {X 0,Y 469.035,Z 1129.634,A -85,B 0,C 180,E1 7184.656,E2 7184.656} C_VEL
LIN {X 0,Y 467.553,Z 1147.087,A -85,B 0,C 180,E1 7187.89,E2 7187.89} C_VEL
LIN {X 0,Y 466.701,Z 1160.075,A -85,B 0,C 180,E1 7191.634,E2 7191.634} C_VEL
LIN {X 0,Y 466.304,Z 1167.203,A -85,B 0,C 180,E1 7195.359,E2 7195.359} C_VEL
LIN {X 0,Y 466.169,Z 1169.211,A -85,B 0,C 180,E1 7198.145,E2 7198.145} C_VEL
LIN {X 0,Y 466.28,Z 1167.59,A -85,B 0,C 180,E1 7201.854,E2 7201.854} C_VEL
LIN {X 0,Y 466.495,Z 1160.937,A -85,B 0,C 180,E1 7205.568,E2 7205.568} C_VEL
LIN {X 0,Y 467.116,Z 1148.613,A -85,B 0,C 180,E1 7209.295,E2 7209.295} C_VEL
LIN {X 0,Y 468.219,Z 1131.831,A -85,B 0,C 180,E1 7212.564,E2 7212.564} C_VEL
LIN {X 0,Y 469.772,Z 1110.213,A -85,B 0,C 180,E1 7215.473,E2 7215.473} C_VEL
LIN {X 0,Y 471.668,Z 1083.612,A -85,B 0,C 180,E1 7217.933,E2 7217.933} C_VEL
LIN {X 0,Y 473.252,Z 1054.011,A -85,B 0,C 180,E1 7219.724,E2 7219.724} C_VEL
LIN {X 0,Y 474.202,Z 1023.443,A -85,B 0,C 180,E1 7220.785,E2 7220.785} C_VEL
LIN {X 0,Y 472.814,Z 1012.914,A -85,B 0,C 180,E1 7221.072,E2 7221.072} C_VEL
LIN {X 0,Y 465.021,Z 989.03,A -85,B 0,C 180,E1 7222.028,E2 7222.028} C_VEL
LIN {X 0,Y 464.732,Z 989.03,A -85,B 0,C 180,E1 7228.742,E2 7228.742} C_VEL
LIN {X 0,Y 464.619,Z 989.03,A -85,B 0,C 180,E1 7233.511,E2 7233.511} C_VEL
LIN {X 0,Y 464.448,Z 989.03,A -85,B 0,C 180,E1 7240.524,E2 7240.524} C_VEL
LIN {X 0,Y 464.587,Z 989.03,A -85,B 0,C 180,E1 7246.986,E2 7246.986} C_VEL
LIN {X 0,Y 464.626,Z 989.03,A -85,B 0,C 180,E1 7251.891,E2 7251.891} C_VEL
LIN {X 0,Y 464.685,Z 989.193,A -85,B 0,C 180,E1 7255.851,E2 7255.851} C_VEL
LIN {X 0,Y 483.009,Z 1030.995,A -85,B 0,C 180,E1 7258.087,E2 7258.087} C_VEL
LIN {X 0,Y 481.53,Z 1067.746,A -85,B 0,C 180,E1 7259.187,E2 7259.187} C_VEL
LIN {X 0,Y 479.027,Z 1102.055,A -85,B 0,C 180,E1 7260.899,E2 7260.899} C_VEL
LIN {X 0,Y 475.854,Z 1134.639,A -85,B 0,C 180,E1 7263.294,E2 7263.294} C_VEL
LIN {X 0,Y 472.612,Z 1164.507,A -85,B 0,C 180,E1 7266.348,E2 7266.348} C_VEL
LIN {X 0,Y 469.666,Z 1190.896,A -85,B 0,C 180,E1 7270.035,E2 7270.035} C_VEL
LIN {X 0,Y 467.534,Z 1211.861,A -85,B 0,C 180,E1 7274.073,E2 7274.073} C_VEL
LIN {X 0,Y 466.327,Z 1227.537,A -85,B 0,C 180,E1 7278.328,E2 7278.328} C_VEL
LIN {X 0,Y 465.858,Z 1237.785,A -85,B 0,C 180,E1 7282.552,E2 7282.552} C_VEL
LIN {X 0,Y 465.748,Z 1242.893,A -85,B 0,C 180,E1 7286.281,E2 7286.281} C_VEL
LIN {X 0,Y 465.643,Z 1244.613,A -85,B 0,C 180,E1 7289.996,E2 7289.996} C_VEL
LIN {X 0,Y 465.799,Z 1241.854,A -85,B 0,C 180,E1 7294.642,E2 7294.642} C_VEL
LIN {X 0,Y 466.056,Z 1233.637,A -85,B 0,C 180,E1 7299.313,E2 7299.313} C_VEL
LIN {X 0,Y 466.854,Z 1220.66,A -85,B 0,C 180,E1 7303.653,E2 7303.653} C_VEL
LIN {X 0,Y 468.418,Z 1202.16,A -85,B 0,C 180,E1 7307.875,E2 7307.875} C_VEL
LIN {X 0,Y 470.91,Z 1178.988,A -85,B 0,C 180,E1 7311.683,E2 7311.683} C_VEL
LIN {X 0,Y 474.038,Z 1151.663,A -85,B 0,C 180,E1 7314.998,E2 7314.998} C_VEL
LIN {X 0,Y 477.428,Z 1119.035,A -85,B 0,C 180,E1 7317.865,E2 7317.865} C_VEL
LIN {X 0,Y 480.29,Z 1085.69,A -85,B 0,C 180,E1 7319.916,E2 7319.916} C_VEL
LIN {X 0,Y 482.424,Z 1049.692,A -85,B 0,C 180,E1 7321.353,E2 7321.353} C_VEL
LIN {X 0,Y 482.725,Z 1029.472,A -85,B 0,C 180,E1 7321.878,E2 7321.878} C_VEL
LIN {X 0,Y 464.711,Z 989.03,A -85,B 0,C 180,E1 7324.156,E2 7324.156} C_VEL
LIN {X 0,Y 464.455,Z 989.03,A -85,B 0,C 180,E1 7330.523,E2 7330.523} C_VEL
LIN {X 0,Y 464.579,Z 989.03,A -85,B 0,C 180,E1 7336.995,E2 7336.995} C_VEL
LIN {X 0,Y 464.622,Z 989.03,A -85,B 0,C 180,E1 7341.899,E2 7341.899} C_VEL
LIN {X 0,Y 464.617,Z 989.03,A -85,B 0,C 180,E1 7348.693,E2 7348.693} C_VEL
LIN {X 0,Y 464.894,Z 989.03,A -85,B 0,C 180,E1 7355.343,E2 7355.343} C_VEL
LIN {X 0,Y 465.014,Z 989.03,A -85,B 0,C 180,E1 7361.066,E2 7361.066} C_VEL
LIN {X 0,Y 465.215,Z 989.03,A -85,B 0,C 180,E1 7366.877,E2 7366.877} C_VEL
LIN {X 0,Y 465.279,Z 989.03,A -85,B 0,C 180,E1 7372.652,E2 7372.652} C_VEL
LIN {X 0,Y 465.424,Z 989.03,A -85,B 0,C 180,E1 7378.142,E2 7378.142} C_VEL
LIN {X 0,Y 465.397,Z 989.03,A -85,B 0,C 180,E1 7383.718,E2 7383.718} C_VEL
LIN {X 0,Y 465.198,Z 989.03,A -85,B 0,C 180,E1 7389.334,E2 7389.334} C_VEL
LIN {X 0,Y 465.039,Z 989.03,A -85,B 0,C 180,E1 7395.046,E2 7395.046} C_VEL
LIN {X 0,Y 464.939,Z 989.03,A -85,B 0,C 180,E1 7400.916,E2 7400.916} C_VEL
LIN {X 0,Y 464.767,Z 989.03,A -85,B 0,C 180,E1 7407.035,E2 7407.035} C_VEL
LIN {X 0,Y 464.603,Z 989.03,A -85,B 0,C 180,E1 7413.513,E2 7413.513} C_VEL
LIN {X 0,Y 464.605,Z 989.03,A -85,B 0,C 180,E1 7418.788,E2 7418.788} C_VEL
LIN {X 0,Y 464.537,Z 989.03,A -85,B 0,C 180,E1 7424.389,E2 7424.389} C_VEL
LIN {X 0,Y 464.575,Z 989.157,A -85,B 0,C 180,E1 7428.489,E2 7428.489} C_VEL
LIN {X 0,Y 475.754,Z 1022.905,A -85,B 0,C 180,E1 7431.746,E2 7431.746} C_VEL
LIN {X 0,Y 487.423,Z 1040.843,A -85,B 0,C 180,E1 7433.005,E2 7433.005} C_VEL
LIN {X 0,Y 486.691,Z 1071.454,A -85,B 0,C 180,E1 7433.606,E2 7433.606} C_VEL
LIN {X 0,Y 482.248,Z 1088.348,A -85,B 0,C 180,E1 7433.832,E2 7433.832} C_VEL
LIN {X 0,Y 478.362,Z 1100.843,A -85,B 0,C 180,E1 7434.062,E2 7434.062} C_VEL
LIN {X 0,Y 477.752,Z 1104.974,A -85,B 0,C 180,E1 7434.204,E2 7434.204} C_VEL
LIN {X 0,Y 474.425,Z 1144.874,A -85,B 0,C 180,E1 7436.193,E2 7436.193} C_VEL
LIN {X 0,Y 470.482,Z 1183.483,A -85,B 0,C 180,E1 7438.949,E2 7438.949} C_VEL
LIN {X 0,Y 466.687,Z 1218.369,A -85,B 0,C 180,E1 7442.337,E2 7442.337} C_VEL
LIN {X 0,Y 463.365,Z 1247.18,A -85,B 0,C 180,E1 7446.076,E2 7446.076} C_VEL
LIN {X 0,Y 460.681,Z 1270.971,A -85,B 0,C 180,E1 7450.385,E2 7450.385} C_VEL
LIN {X 0,Y 458.888,Z 1290.386,A -85,B 0,C 180,E1 7455.24,E2 7455.24} C_VEL
LIN {X 0,Y 458.09,Z 1303.707,A -85,B 0,C 180,E1 7460.044,E2 7460.044} C_VEL
LIN {X 0,Y 457.738,Z 1310.979,A -85,B 0,C 180,E1 7464.328,E2 7464.328} C_VEL
LIN {X 0,Y 457.715,Z 1314.108,A -85,B 0,C 180,E1 7468.114,E2 7468.114} C_VEL
LIN {X 0,Y 457.766,Z 1314.109,A -85,B 0,C 180,E1 7471.893,E2 7471.893} C_VEL
LIN {X 0,Y 457.844,Z 1309.684,A -85,B 0,C 180,E1 7476.628,E2 7476.628} C_VEL
LIN {X 0,Y 458.195,Z 1300.248,A -85,B 0,C 180,E1 7481.401,E2 7481.401} C_VEL
LIN {X 0,Y 459.331,Z 1285.251,A -85,B 0,C 180,E1 7486.219,E2 7486.219} C_VEL
LIN {X 0,Y 461.449,Z 1263.602,A -85,B 0,C 180,E1 7491.087,E2 7491.087} C_VEL
LIN {X 0,Y 464.077,Z 1241.386,A -85,B 0,C 180,E1 7494.792,E2 7494.792} C_VEL
LIN {X 0,Y 467.016,Z 1213.359,A -85,B 0,C 180,E1 7498.074,E2 7498.074} C_VEL
LIN {X 0,Y 470.338,Z 1178.623,A -85,B 0,C 180,E1 7501.147,E2 7501.147} C_VEL
LIN {X 0,Y 473.583,Z 1139.017,A -85,B 0,C 180,E1 7503.691,E2 7503.691} C_VEL
LIN {X 0,Y 476.245,Z 1096.031,A -85,B 0,C 180,E1 7505.581,E2 7505.581} C_VEL
LIN {X 0,Y 478.292,Z 1052.792,A -85,B 0,C 180,E1 7506.705,E2 7506.705} C_VEL
LIN {X 0,Y 477.714,Z 1041.944,A -85,B 0,C 180,E1 7506.934,E2 7506.934} C_VEL
LIN {X 0,Y 464.963,Z 1019.337,A -85,B 0,C 180,E1 7508.125,E2 7508.125} C_VEL
LIN {X 0,Y 460.551,Z 1004.752,A -85,B 0,C 180,E1 7508.876,E2 7508.876} C_VEL
LIN {X 0,Y 456.745,Z 989.03,A -85,B 0,C 180,E1 7510.26,E2 7510.26} C_VEL
LIN {X 0,Y 456.616,Z 989.03,A -85,B 0,C 180,E1 7516.647,E2 7516.647} C_VEL
LIN {X 0,Y 456.598,Z 989.03,A -85,B 0,C 180,E1 7523.497,E2 7523.497} C_VEL
LIN {X 0,Y 456.786,Z 989.03,A -85,B 0,C 180,E1 7530.296,E2 7530.296} C_VEL
LIN {X 0,Y 456.932,Z 989.03,A -85,B 0,C 180,E1 7535.225,E2 7535.225} C_VEL
LIN {X 0,Y 467.054,Z 1019.498,A -85,B 0,C 180,E1 7536.616,E2 7536.616} C_VEL
LIN {X 0,Y 466.589,Z 1052.031,A -85,B 0,C 180,E1 7537.548,E2 7537.548} C_VEL
LIN {X 0,Y 465.288,Z 1080.656,A -85,B 0,C 180,E1 7539.1,E2 7539.1} C_VEL
LIN {X 0,Y 463.456,Z 1107.257,A -85,B 0,C 180,E1 7541.368,E2 7541.368} C_VEL
LIN {X 0,Y 461.713,Z 1129.147,A -85,B 0,C 180,E1 7544.115,E2 7544.115} C_VEL
LIN {X 0,Y 460.015,Z 1147.452,A -85,B 0,C 180,E1 7547.448,E2 7547.448} C_VEL
LIN {X 0,Y 459.084,Z 1160.216,A -85,B 0,C 180,E1 7551.018,E2 7551.018} C_VEL
LIN {X 0,Y 458.658,Z 1167.313,A -85,B 0,C 180,E1 7554.335,E2 7554.335} C_VEL
LIN {X 0,Y 458.41,Z 1170.582,A -85,B 0,C 180,E1 7558.113,E2 7558.113} C_VEL
LIN {X 0,Y 458.52,Z 1168.915,A -85,B 0,C 180,E1 7561.886,E2 7561.886} C_VEL
LIN {X 0,Y 458.741,Z 1162.224,A -85,B 0,C 180,E1 7565.663,E2 7565.663} C_VEL
LIN {X 0,Y 459.416,Z 1149.835,A -85,B 0,C 180,E1 7569.452,E2 7569.452} C_VEL
LIN {X 0,Y 460.6,Z 1133.007,A -85,B 0,C 180,E1 7572.775,E2 7572.775} C_VEL
LIN {X 0,Y 462.255,Z 1111.357,A -85,B 0,C 180,E1 7575.731,E2 7575.731} C_VEL
LIN {X 0,Y 464.237,Z 1084.755,A -85,B 0,C 180,E1 7578.231,E2 7578.231} C_VEL
LIN {X 0,Y 465.917,Z 1054.994,A -85,B 0,C 180,E1 7580.059,E2 7580.059} C_VEL
LIN {X 0,Y 466.918,Z 1022.609,A -85,B 0,C 180,E1 7581.179,E2 7581.179} C_VEL
LIN {X 0,Y 464.055,Z 1010.182,A -85,B 0,C 180,E1 7581.579,E2 7581.579} C_VEL
LIN {X 0,Y 457.074,Z 989.03,A -85,B 0,C 180,E1 7582.407,E2 7582.407} C_VEL
LIN {X 0,Y 456.807,Z 989.03,A -85,B 0,C 180,E1 7587.545,E2 7587.545} C_VEL
LIN {X 0,Y 456.623,Z 989.03,A -85,B 0,C 180,E1 7594.283,E2 7594.283} C_VEL
LIN {X 0,Y 456.564,Z 989.03,A -85,B 0,C 180,E1 7600.512,E2 7600.512} C_VEL
LIN {X 0,Y 456.683,Z 989.03,A -85,B 0,C 180,E1 7606.627,E2 7606.627} C_VEL
LIN {X 0,Y 456.667,Z 989.03,A -85,B 0,C 180,E1 7613.496,E2 7613.496} C_VEL
LIN {X 0,Y 456.837,Z 989.817,A -85,B 0,C 180,E1 7615.183,E2 7615.183} C_VEL
LIN {X 0,Y 476.285,Z 1033.213,A -85,B 0,C 180,E1 7617.622,E2 7617.622} C_VEL
LIN {X 0,Y 474.595,Z 1071.086,A -85,B 0,C 180,E1 7618.812,E2 7618.812} C_VEL
LIN {X 0,Y 471.807,Z 1106.237,A -85,B 0,C 180,E1 7620.671,E2 7620.671} C_VEL
LIN {X 0,Y 468.532,Z 1137.38,A -85,B 0,C 180,E1 7623.053,E2 7623.053} C_VEL
LIN {X 0,Y 465.217,Z 1166.099,A -85,B 0,C 180,E1 7626.075,E2 7626.075} C_VEL
LIN {X 0,Y 462.198,Z 1191.487,A -85,B 0,C 180,E1 7629.698,E2 7629.698} C_VEL
LIN {X 0,Y 459.865,Z 1212.461,A -85,B 0,C 180,E1 7633.8,E2 7633.8} C_VEL
LIN {X 0,Y 458.564,Z 1228.137,A -85,B 0,C 180,E1 7638.127,E2 7638.127} C_VEL
LIN {X 0,Y 458.019,Z 1238.386,A -85,B 0,C 180,E1 7642.423,E2 7642.423} C_VEL
LIN {X 0,Y 457.873,Z 1243.495,A -85,B 0,C 180,E1 7646.217,E2 7646.217} C_VEL
LIN {X 0,Y 457.767,Z 1245.214,A -85,B 0,C 180,E1 7649.996,E2 7649.996} C_VEL
LIN {X 0,Y 457.928,Z 1242.457,A -85,B 0,C 180,E1 7654.722,E2 7654.722} C_VEL
LIN {X 0,Y 458.219,Z 1234.243,A -85,B 0,C 180,E1 7659.474,E2 7659.474} C_VEL
LIN {X 0,Y 459.208,Z 1220.222,A -85,B 0,C 180,E1 7664.18,E2 7664.18} C_VEL
LIN {X 0,Y 461.09,Z 1200.62,A -85,B 0,C 180,E1 7668.585,E2 7668.585} C_VEL
LIN {X 0,Y 463.917,Z 1176.428,A -85,B 0,C 180,E1 7672.499,E2 7672.499} C_VEL
LIN {X 0,Y 467.319,Z 1148.068,A -85,B 0,C 180,E1 7675.84,E2 7675.84} C_VEL
LIN {X 0,Y 470.648,Z 1117.765,A -85,B 0,C 180,E1 7678.449,E2 7678.449} C_VEL
LIN {X 0,Y 473.743,Z 1083.133,A -85,B 0,C 180,E1 7680.549,E2 7680.549} C_VEL
LIN {X 0,Y 475.961,Z 1046.001,A -85,B 0,C 180,E1 7681.964,E2 7681.964} C_VEL
LIN {X 0,Y 475.941,Z 1031.679,A -85,B 0,C 180,E1 7682.348,E2 7682.348} C_VEL
LIN {X 0,Y 456.767,Z 989.03,A -85,B 0,C 180,E1 7684.806,E2 7684.806} C_VEL
LIN {X 0,Y 456.573,Z 989.03,A -85,B 0,C 180,E1 7691.374,E2 7691.374} C_VEL
LIN {X 0,Y 456.668,Z 989.03,A -85,B 0,C 180,E1 7696.629,E2 7696.629} C_VEL
LIN {X 0,Y 456.681,Z 989.03,A -85,B 0,C 180,E1 7702.466,E2 7702.466} C_VEL
LIN {X 0,Y 456.68,Z 989.03,A -85,B 0,C 180,E1 7709.213,E2 7709.213} C_VEL
LIN {X 0,Y 456.874,Z 989.03,A -85,B 0,C 180,E1 7714.574,E2 7714.574} C_VEL
LIN {X 0,Y 457.085,Z 989.03,A -85,B 0,C 180,E1 7720.724,E2 7720.724} C_VEL
LIN {X 0,Y 457.312,Z 989.03,A -85,B 0,C 180,E1 7726.646,E2 7726.646} C_VEL
LIN {X 0,Y 457.353,Z 989.03,A -85,B 0,C 180,E1 7732.644,E2 7732.644} C_VEL
LIN {X 0,Y 457.521,Z 989.03,A -85,B 0,C 180,E1 7738.11,E2 7738.11} C_VEL
LIN {X 0,Y 457.488,Z 989.03,A -85,B 0,C 180,E1 7743.783,E2 7743.783} C_VEL
LIN {X 0,Y 457.286,Z 989.03,A -85,B 0,C 180,E1 7749.497,E2 7749.497} C_VEL
LIN {X 0,Y 457.104,Z 989.03,A -85,B 0,C 180,E1 7755.313,E2 7755.313} C_VEL
LIN {X 0,Y 456.979,Z 989.03,A -85,B 0,C 180,E1 7761.298,E2 7761.298} C_VEL
LIN {X 0,Y 456.824,Z 989.03,A -85,B 0,C 180,E1 7767.545,E2 7767.545} C_VEL
LIN {X 0,Y 456.65,Z 989.03,A -85,B 0,C 180,E1 7774.301,E2 7774.301} C_VEL
LIN {X 0,Y 456.688,Z 989.03,A -85,B 0,C 180,E1 7780.542,E2 7780.542} C_VEL
LIN {X 0,Y 456.62,Z 989.03,A -85,B 0,C 180,E1 7787.098,E2 7787.098} C_VEL
LIN {X 0,Y 456.641,Z 989.218,A -85,B 0,C 180,E1 7787.8,E2 7787.8} C_VEL
LIN {X 0,Y 467.572,Z 1021.778,A -85,B 0,C 180,E1 7791.037,E2 7791.037} C_VEL
LIN {X 0,Y 478.802,Z 1041.642,A -85,B 0,C 180,E1 7792.356,E2 7792.356} C_VEL
LIN {X 0,Y 480.837,Z 1044.412,A -85,B 0,C 180,E1 7792.563,E2 7792.563} C_VEL
LIN {X 0,Y 479.077,Z 1087.167,A -85,B 0,C 180,E1 7793.567,E2 7793.567} C_VEL
LIN {X 0,Y 477.752,Z 1104.974,A -85,B 0,C 180,E1 7794.204,E2 7794.204} C_VEL
LIN {X 0,Y 473.004,Z 1121.496,A -85,B 0,C 180,E1 7794.707,E2 7794.707} C_VEL
LIN {X 0,Y 468.061,Z 1137.391,A -85,B 0,C 180,E1 7795.323,E2 7795.323} C_VEL
LIN {X 0,Y 463.992,Z 1175.779,A -85,B 0,C 180,E1 7797.952,E2 7797.952} C_VEL
LIN {X 0,Y 459.996,Z 1210.546,A -85,B 0,C 180,E1 7801.199,E2 7801.199} C_VEL
LIN {X 0,Y 456.353,Z 1241.315,A -85,B 0,C 180,E1 7804.988,E2 7804.988} C_VEL
LIN {X 0,Y 453.487,Z 1266.234,A -85,B 0,C 180,E1 7809.083,E2 7809.083} C_VEL
LIN {X 0,Y 451.478,Z 1285.291,A -85,B 0,C 180,E1 7813.498,E2 7813.498} C_VEL
LIN {X 0,Y 450.407,Z 1299.079,A -85,B 0,C 180,E1 7817.917,E2 7817.917} C_VEL
LIN {X 0,Y 449.975,Z 1308.226,A -85,B 0,C 180,E1 7822.295,E2 7822.295} C_VEL
LIN {X 0,Y 449.805,Z 1312.93,A -85,B 0,C 180,E1 7826.156,E2 7826.156} C_VEL
LIN {X 0,Y 449.847,Z 1314.5,A -85,B 0,C 180,E1 7830.004,E2 7830.004} C_VEL
LIN {X 0,Y 449.796,Z 1312.933,A -85,B 0,C 180,E1 7833.851,E2 7833.851} C_VEL
LIN {X 0,Y 450.064,Z 1306.211,A -85,B 0,C 180,E1 7838.853,E2 7838.853} C_VEL
LIN {X 0,Y 450.816,Z 1293.942,A -85,B 0,C 180,E1 7843.91,E2 7843.91} C_VEL
LIN {X 0,Y 452.29,Z 1277.163,A -85,B 0,C 180,E1 7848.55,E2 7848.55} C_VEL
LIN {X 0,Y 454.507,Z 1257.757,A -85,B 0,C 180,E1 7852.451,E2 7852.451} C_VEL
LIN {X 0,Y 457.422,Z 1230.202,A -85,B 0,C 180,E1 7856.346,E2 7856.346} C_VEL
LIN {X 0,Y 460.955,Z 1196.471,A -85,B 0,C 180,E1 7859.88,E2 7859.88} C_VEL
LIN {X 0,Y 464.456,Z 1158.839,A -85,B 0,C 180,E1 7862.781,E2 7862.781} C_VEL
LIN {X 0,Y 467.6,Z 1118.077,A -85,B 0,C 180,E1 7865.023,E2 7865.023} C_VEL
LIN {X 0,Y 470.151,Z 1076.222,A -85,B 0,C 180,E1 7866.547,E2 7866.547} C_VEL
LIN {X 0,Y 470.845,Z 1045.369,A -85,B 0,C 180,E1 7867.272,E2 7867.272} C_VEL
LIN {X 0,Y 458.565,Z 1022.737,A -85,B 0,C 180,E1 7868.508,E2 7868.508} C_VEL
LIN {X 0,Y 452.414,Z 1002.737,A -85,B 0,C 180,E1 7869.489,E2 7869.489} C_VEL
LIN {X 0,Y 448.794,Z 989.03,A -85,B 0,C 180,E1 7870.744,E2 7870.744} C_VEL
LIN {X 0,Y 448.642,Z 989.03,A -85,B 0,C 180,E1 7877.736,E2 7877.736} C_VEL
LIN {X 0,Y 448.667,Z 989.03,A -85,B 0,C 180,E1 7883.831,E2 7883.831} C_VEL
LIN {X 0,Y 448.85,Z 989.03,A -85,B 0,C 180,E1 7889.717,E2 7889.717} C_VEL
LIN {X 0,Y 449.002,Z 989.687,A -85,B 0,C 180,E1 7894.651,E2 7894.651} C_VEL
LIN {X 0,Y 459.876,Z 1021.114,A -85,B 0,C 180,E1 7896.227,E2 7896.227} C_VEL
LIN {X 0,Y 459.387,Z 1054.708,A -85,B 0,C 180,E1 7897.229,E2 7897.229} C_VEL
LIN {X 0,Y 457.958,Z 1083.858,A -85,B 0,C 180,E1 7898.876,E2 7898.876} C_VEL
LIN {X 0,Y 455.996,Z 1109.904,A -85,B 0,C 180,E1 7901.177,E2 7901.177} C_VEL
LIN {X 0,Y 454.11,Z 1132.188,A -85,B 0,C 180,E1 7904.089,E2 7904.089} C_VEL
LIN {X 0,Y 452.368,Z 1149.96,A -85,B 0,C 180,E1 7907.477,E2 7907.477} C_VEL
LIN {X 0,Y 451.415,Z 1161.788,A -85,B 0,C 180,E1 7910.918,E2 7910.918} C_VEL
LIN {X 0,Y 450.917,Z 1168.721,A -85,B 0,C 180,E1 7914.238,E2 7914.238} C_VEL
LIN {X 0,Y 450.634,Z 1171.959,A -85,B 0,C 180,E1 7918.081,E2 7918.081} C_VEL
LIN {X 0,Y 450.736,Z 1170.243,A -85,B 0,C 180,E1 7921.918,E2 7921.918} C_VEL
LIN {X 0,Y 450.99,Z 1163.497,A -85,B 0,C 180,E1 7925.76,E2 7925.76} C_VEL
LIN {X 0,Y 451.722,Z 1151.056,A -85,B 0,C 180,E1 7929.614,E2 7929.614} C_VEL
LIN {X 0,Y 452.995,Z 1134.183,A -85,B 0,C 180,E1 7932.993,E2 7932.993} C_VEL
LIN {X 0,Y 454.872,Z 1111.577,A -85,B 0,C 180,E1 7936.104,E2 7936.104} C_VEL
LIN {X 0,Y 456.837,Z 1085.881,A -85,B 0,C 180,E1 7938.536,E2 7938.536} C_VEL
LIN {X 0,Y 458.573,Z 1056.159,A -85,B 0,C 180,E1 7940.394,E2 7940.394} C_VEL
LIN {X 0,Y 459.621,Z 1026.028,A -85,B 0,C 180,E1 7941.484,E2 7941.484} C_VEL
LIN {X 0,Y 458.245,Z 1016.212,A -85,B 0,C 180,E1 7941.776,E2 7941.776} C_VEL
LIN {X 0,Y 449.101,Z 989.03,A -85,B 0,C 180,E1 7942.91,E2 7942.91} C_VEL
LIN {X 0,Y 448.77,Z 989.03,A -85,B 0,C 180,E1 7949.032,E2 7949.032} C_VEL
LIN {X 0,Y 448.651,Z 989.03,A -85,B 0,C 180,E1 7954.872,E2 7954.872} C_VEL
LIN {X 0,Y 448.645,Z 989.03,A -85,B 0,C 180,E1 7959.719,E2 7959.719} C_VEL
LIN {X 0,Y 448.668,Z 989.03,A -85,B 0,C 180,E1 7965.059,E2 7965.059} C_VEL
LIN {X 0,Y 448.77,Z 989.03,A -85,B 0,C 180,E1 7970.655,E2 7970.655} C_VEL
LIN {X 0,Y 448.854,Z 989.629,A -85,B 0,C 180,E1 7974.458,E2 7974.458} C_VEL
LIN {X 0,Y 469.58,Z 1035.356,A -85,B 0,C 180,E1 7977.141,E2 7977.141} C_VEL
LIN {X 0,Y 467.764,Z 1072.933,A -85,B 0,C 180,E1 7978.37,E2 7978.37} C_VEL
LIN {X 0,Y 464.962,Z 1106.398,A -85,B 0,C 180,E1 7980.167,E2 7980.167} C_VEL
LIN {X 0,Y 461.435,Z 1138.355,A -85,B 0,C 180,E1 7982.644,E2 7982.644} C_VEL
LIN {X 0,Y 457.874,Z 1167.058,A -85,B 0,C 180,E1 7985.715,E2 7985.715} C_VEL
LIN {X 0,Y 454.524,Z 1193.48,A -85,B 0,C 180,E1 7989.594,E2 7989.594} C_VEL
LIN {X 0,Y 452.088,Z 1214.099,A -85,B 0,C 180,E1 7993.763,E2 7993.763} C_VEL
LIN {X 0,Y 450.684,Z 1230.171,A -85,B 0,C 180,E1 7998.407,E2 7998.407} C_VEL
LIN {X 0,Y 450.17,Z 1238.988,A -85,B 0,C 180,E1 8002.29,E2 8002.29} C_VEL
LIN {X 0,Y 450.016,Z 1244.095,A -85,B 0,C 180,E1 8006.151,E2 8006.151} C_VEL
LIN {X 0,Y 449.911,Z 1245.813,A -85,B 0,C 180,E1 8009.996,E2 8009.996} C_VEL
LIN {X 0,Y 450.077,Z 1243.059,A -85,B 0,C 180,E1 8014.805,E2 8014.805} C_VEL
LIN {X 0,Y 450.41,Z 1234.848,A -85,B 0,C 180,E1 8019.64,E2 8019.64} C_VEL
LIN {X 0,Y 451.411,Z 1221.586,A -85,B 0,C 180,E1 8024.215,E2 8024.215} C_VEL
LIN {X 0,Y 453.356,Z 1202.707,A -85,B 0,C 180,E1 8028.62,E2 8028.62} C_VEL
LIN {X 0,Y 456.272,Z 1179.136,A -85,B 0,C 180,E1 8032.575,E2 8032.575} C_VEL
LIN {X 0,Y 459.93,Z 1151.072,A -85,B 0,C 180,E1 8036.026,E2 8036.026} C_VEL
LIN {X 0,Y 463.507,Z 1120.188,A -85,B 0,C 180,E1 8038.779,E2 8038.779} C_VEL
LIN {X 0,Y 466.728,Z 1086.323,A -85,B 0,C 180,E1 8040.907,E2 8040.907} C_VEL
LIN {X 0,Y 469.158,Z 1049.357,A -85,B 0,C 180,E1 8042.396,E2 8042.396} C_VEL
LIN {X 0,Y 469.287,Z 1034.011,A -85,B 0,C 180,E1 8042.822,E2 8042.822} C_VEL
LIN {X 0,Y 448.801,Z 989.03,A -85,B 0,C 180,E1 8045.527,E2 8045.527} C_VEL
LIN {X 0,Y 448.633,Z 989.03,A -85,B 0,C 180,E1 8052.273,E2 8052.273} C_VEL
LIN {X 0,Y 448.708,Z 989.03,A -85,B 0,C 180,E1 8057.735,E2 8057.735} C_VEL
LIN {X 0,Y 448.734,Z 989.03,A -85,B 0,C 180,E1 8063.807,E2 8063.807} C_VEL
LIN {X 0,Y 448.781,Z 989.03,A -85,B 0,C 180,E1 8069.713,E2 8069.713} C_VEL
LIN {X 0,Y 449.004,Z 989.03,A -85,B 0,C 180,E1 8076.217,E2 8076.217} C_VEL
LIN {X 0,Y 449.236,Z 989.03,A -85,B 0,C 180,E1 8082.405,E2 8082.405} C_VEL
LIN {X 0,Y 449.382,Z 989.03,A -85,B 0,C 180,E1 8088.378,E2 8088.378} C_VEL
LIN {X 0,Y 449.556,Z 989.03,A -85,B 0,C 180,E1 8094.221,E2 8094.221} C_VEL
LIN {X 0,Y 449.763,Z 989.03,A -85,B 0,C 180,E1 8100,E2 8100} C_VEL
LIN {X 0,Y 449.58,Z 989.03,A -85,B 0,C 180,E1 8105.779,E2 8105.779} C_VEL
LIN {X 0,Y 449.321,Z 989.03,A -85,B 0,C 180,E1 8111.625,E2 8111.625} C_VEL
LIN {X 0,Y 449.123,Z 989.03,A -85,B 0,C 180,E1 8117.601,E2 8117.601} C_VEL
LIN {X 0,Y 448.958,Z 989.03,A -85,B 0,C 180,E1 8123.786,E2 8123.786} C_VEL
LIN {X 0,Y 448.774,Z 989.03,A -85,B 0,C 180,E1 8130.289,E2 8130.289} C_VEL
LIN {X 0,Y 448.767,Z 989.03,A -85,B 0,C 180,E1 8137.246,E2 8137.246} C_VEL
LIN {X 0,Y 448.712,Z 989.03,A -85,B 0,C 180,E1 8142.284,E2 8142.284} C_VEL
LIN {X 0,Y 448.736,Z 989.325,A -85,B 0,C 180,E1 8147.103,E2 8147.103} C_VEL
LIN {X 0,Y 459.224,Z 1020.242,A -85,B 0,C 180,E1 8150.273,E2 8150.273} C_VEL
LIN {X 0,Y 470.489,Z 1042.319,A -85,B 0,C 180,E1 8151.7,E2 8151.7} C_VEL
LIN {X 0,Y 474.194,Z 1047.877,A -85,B 0,C 180,E1 8152.1,E2 8152.1} C_VEL
LIN {X 0,Y 471.978,Z 1091.449,A -85,B 0,C 180,E1 8153.226,E2 8153.226} C_VEL
LIN {X 0,Y 468.719,Z 1130.866,A -85,B 0,C 180,E1 8154.965,E2 8154.965} C_VEL
LIN {X 0,Y 468.061,Z 1137.391,A -85,B 0,C 180,E1 8155.323,E2 8155.323} C_VEL
LIN {X 0,Y 462.814,Z 1153.021,A -85,B 0,C 180,E1 8156.066,E2 8156.066} C_VEL
LIN {X 0,Y 457.596,Z 1168.105,A -85,B 0,C 180,E1 8156.952,E2 8156.952} C_VEL
LIN {X 0,Y 453.219,Z 1204.025,A -85,B 0,C 180,E1 8160.178,E2 8160.178} C_VEL
LIN {X 0,Y 449.204,Z 1236.575,A -85,B 0,C 180,E1 8164.109,E2 8164.109} C_VEL
LIN {X 0,Y 446.027,Z 1263.203,A -85,B 0,C 180,E1 8168.371,E2 8168.371} C_VEL
LIN {X 0,Y 443.925,Z 1283.358,A -85,B 0,C 180,E1 8172.7,E2 8172.7} C_VEL
LIN {X 0,Y 442.653,Z 1297.777,A -85,B 0,C 180,E1 8177.201,E2 8177.201} C_VEL
LIN {X 0,Y 442.079,Z 1308.222,A -85,B 0,C 180,E1 8182.156,E2 8182.156} C_VEL
LIN {X 0,Y 441.899,Z 1312.926,A -85,B 0,C 180,E1 8186.088,E2 8186.088} C_VEL
LIN {X 0,Y 441.946,Z 1314.5,A -85,B 0,C 180,E1 8190.004,E2 8190.004} C_VEL
LIN {X 0,Y 441.893,Z 1312.929,A -85,B 0,C 180,E1 8193.92,E2 8193.92} C_VEL
LIN {X 0,Y 442.186,Z 1306.456,A -85,B 0,C 180,E1 8198.883,E2 8198.883} C_VEL
LIN {X 0,Y 442.989,Z 1293.937,A -85,B 0,C 180,E1 8204.161,E2 8204.161} C_VEL
LIN {X 0,Y 444.452,Z 1278.245,A -85,B 0,C 180,E1 8208.569,E2 8208.569} C_VEL
LIN {X 0,Y 446.841,Z 1255.48,A -85,B 0,C 180,E1 8212.857,E2 8212.857} C_VEL
LIN {X 0,Y 449.889,Z 1227.695,A -85,B 0,C 180,E1 8216.77,E2 8216.77} C_VEL
LIN {X 0,Y 453.409,Z 1194.287,A -85,B 0,C 180,E1 8220.277,E2 8220.277} C_VEL
LIN {X 0,Y 457.031,Z 1156.941,A -85,B 0,C 180,E1 8223.174,E2 8223.174} C_VEL
LIN {X 0,Y 460.331,Z 1116.043,A -85,B 0,C 180,E1 8225.448,E2 8225.448} C_VEL
LIN {X 0,Y 463.073,Z 1073.969,A -85,B 0,C 180,E1 8227.005,E2 8227.005} C_VEL
LIN {X 0,Y 463.404,Z 1047.667,A -85,B 0,C 180,E1 8227.691,E2 8227.691} C_VEL
LIN {X 0,Y 452.04,Z 1025.648,A -85,B 0,C 180,E1 8228.943,E2 8228.943} C_VEL
LIN {X 0,Y 443.436,Z 998.375,A -85,B 0,C 180,E1 8230.39,E2 8230.39} C_VEL
LIN {X 0,Y 440.9,Z 989.03,A -85,B 0,C 180,E1 8231.345,E2 8231.345} C_VEL
LIN {X 0,Y 440.636,Z 989.03,A -85,B 0,C 180,E1 8236.772,E2 8236.772} C_VEL
LIN {X 0,Y 440.712,Z 989.03,A -85,B 0,C 180,E1 8241.963,E2 8241.963} C_VEL
LIN {X 0,Y 440.802,Z 989.03,A -85,B 0,C 180,E1 8246.79,E2 8246.79} C_VEL
LIN {X 0,Y 440.964,Z 989.03,A -85,B 0,C 180,E1 8253.586,E2 8253.586} C_VEL
LIN {X 0,Y 441.078,Z 989.808,A -85,B 0,C 180,E1 8253.979,E2 8253.979} C_VEL
LIN {X 0,Y 451.637,Z 1018.676,A -85,B 0,C 180,E1 8255.639,E2 8255.639} C_VEL
LIN {X 0,Y 452.798,Z 1027.395,A -85,B 0,C 180,E1 8255.93,E2 8255.93} C_VEL
LIN {X 0,Y 452.143,Z 1059.167,A -85,B 0,C 180,E1 8256.971,E2 8256.971} C_VEL
LIN {X 0,Y 450.663,Z 1087.167,A -85,B 0,C 180,E1 8258.646,E2 8258.646} C_VEL
LIN {X 0,Y 448.644,Z 1112.568,A -85,B 0,C 180,E1 8260.984,E2 8260.984} C_VEL
LIN {X 0,Y 446.553,Z 1135.213,A -85,B 0,C 180,E1 8264.064,E2 8264.064} C_VEL
LIN {X 0,Y 444.803,Z 1151.415,A -85,B 0,C 180,E1 8267.261,E2 8267.261} C_VEL
LIN {X 0,Y 443.703,Z 1163.545,A -85,B 0,C 180,E1 8270.877,E2 8270.877} C_VEL
LIN {X 0,Y 443.074,Z 1171.408,A -85,B 0,C 180,E1 8275.116,E2 8275.116} C_VEL
LIN {X 0,Y 442.875,Z 1173.337,A -85,B 0,C 180,E1 8278.047,E2 8278.047} C_VEL
LIN {X 0,Y 442.976,Z 1171.568,A -85,B 0,C 180,E1 8281.952,E2 8281.952} C_VEL
LIN {X 0,Y 443.234,Z 1164.776,A -85,B 0,C 180,E1 8285.862,E2 8285.862} C_VEL
LIN {X 0,Y 444.046,Z 1152.268,A -85,B 0,C 180,E1 8289.782,E2 8289.782} C_VEL
LIN {X 0,Y 445.381,Z 1135.337,A -85,B 0,C 180,E1 8293.219,E2 8293.219} C_VEL
LIN {X 0,Y 447.292,Z 1113.401,A -85,B 0,C 180,E1 8296.295,E2 8296.295} C_VEL
LIN {X 0,Y 449.449,Z 1086.937,A -85,B 0,C 180,E1 8298.853,E2 8298.853} C_VEL
LIN {X 0,Y 451.241,Z 1057.475,A -85,B 0,C 180,E1 8300.728,E2 8300.728} C_VEL
LIN {X 0,Y 452.374,Z 1025.683,A -85,B 0,C 180,E1 8301.885,E2 8301.885} C_VEL
LIN {X 0,Y 448.556,Z 1010.751,A -85,B 0,C 180,E1 8302.418,E2 8302.418} C_VEL
LIN {X 0,Y 441.117,Z 989.03,A -85,B 0,C 180,E1 8303.402,E2 8303.402} C_VEL
LIN {X 0,Y 440.906,Z 989.03,A -85,B 0,C 180,E1 8308.628,E2 8308.628} C_VEL
LIN {X 0,Y 440.724,Z 989.03,A -85,B 0,C 180,E1 8315.594,E2 8315.594} C_VEL
LIN {X 0,Y 440.635,Z 989.03,A -85,B 0,C 180,E1 8321.105,E2 8321.105} C_VEL
LIN {X 0,Y 440.721,Z 989.03,A -85,B 0,C 180,E1 8326.774,E2 8326.774} C_VEL
LIN {X 0,Y 440.881,Z 989.15,A -85,B 0,C 180,E1 8333.695,E2 8333.695} C_VEL
LIN {X 0,Y 462.957,Z 1037.655,A -85,B 0,C 180,E1 8336.654,E2 8336.654} C_VEL
LIN {X 0,Y 460.958,Z 1074.832,A -85,B 0,C 180,E1 8337.918,E2 8337.918} C_VEL
LIN {X 0,Y 457.975,Z 1108.416,A -85,B 0,C 180,E1 8339.773,E2 8339.773} C_VEL
LIN {X 0,Y 454.129,Z 1141.327,A -85,B 0,C 180,E1 8342.406,E2 8342.406} C_VEL
LIN {X 0,Y 450.146,Z 1171.468,A -85,B 0,C 180,E1 8345.801,E2 8345.801} C_VEL
LIN {X 0,Y 446.86,Z 1195.472,A -85,B 0,C 180,E1 8349.486,E2 8349.486} C_VEL
LIN {X 0,Y 444.314,Z 1215.736,A -85,B 0,C 180,E1 8353.724,E2 8353.724} C_VEL
LIN {X 0,Y 442.922,Z 1230.771,A -85,B 0,C 180,E1 8358.2,E2 8358.2} C_VEL
LIN {X 0,Y 442.335,Z 1239.589,A -85,B 0,C 180,E1 8362.153,E2 8362.153} C_VEL
LIN {X 0,Y 442.14,Z 1244.697,A -85,B 0,C 180,E1 8366.082,E2 8366.082} C_VEL
LIN {X 0,Y 442.034,Z 1246.415,A -85,B 0,C 180,E1 8369.996,E2 8369.996} C_VEL
LIN {X 0,Y 442.224,Z 1243.661,A -85,B 0,C 180,E1 8374.89,E2 8374.89} C_VEL
LIN {X 0,Y 442.585,Z 1235.453,A -85,B 0,C 180,E1 8379.812,E2 8379.812} C_VEL
LIN {X 0,Y 443.712,Z 1222.19,A -85,B 0,C 180,E1 8384.467,E2 8384.467} C_VEL
LIN {X 0,Y 445.865,Z 1203.004,A -85,B 0,C 180,E1 8389.006,E2 8389.006} C_VEL
LIN {X 0,Y 449.037,Z 1178.939,A -85,B 0,C 180,E1 8393.083,E2 8393.083} C_VEL
LIN {X 0,Y 452.932,Z 1150.455,A -85,B 0,C 180,E1 8396.592,E2 8396.592} C_VEL
LIN {X 0,Y 456.774,Z 1118.92,A -85,B 0,C 180,E1 8399.397,E2 8399.397} C_VEL
LIN {X 0,Y 460.142,Z 1085.117,A -85,B 0,C 180,E1 8401.503,E2 8401.503} C_VEL
LIN {X 0,Y 462.669,Z 1047.451,A -85,B 0,C 180,E1 8402.985,E2 8402.985} C_VEL
LIN {X 0,Y 462.412,Z 1035.839,A -85,B 0,C 180,E1 8403.343,E2 8403.343} C_VEL
LIN {X 0,Y 442.372,Z 993.68,A -85,B 0,C 180,E1 8405.977,E2 8405.977} C_VEL
LIN {X 0,Y 440.814,Z 989.03,A -85,B 0,C 180,E1 8406.285,E2 8406.285} C_VEL
LIN {X 0,Y 440.624,Z 989.03,A -85,B 0,C 180,E1 8413.227,E2 8413.227} C_VEL
LIN {X 0,Y 440.734,Z 989.03,A -85,B 0,C 180,E1 8419.421,E2 8419.421} C_VEL
LIN {X 0,Y 440.802,Z 989.03,A -85,B 0,C 180,E1 8425.241,E2 8425.241} C_VEL
LIN {X 0,Y 440.919,Z 989.03,A -85,B 0,C 180,E1 8431.373,E2 8431.373} C_VEL
LIN {X 0,Y 441.117,Z 989.03,A -85,B 0,C 180,E1 8437.897,E2 8437.897} C_VEL
LIN {X 0,Y 441.387,Z 989.03,A -85,B 0,C 180,E1 8444.128,E2 8444.128} C_VEL
LIN {X 0,Y 441.541,Z 989.03,A -85,B 0,C 180,E1 8450.162,E2 8450.162} C_VEL
LIN {X 0,Y 441.741,Z 989.03,A -85,B 0,C 180,E1 8456.083,E2 8456.083} C_VEL
LIN {X 0,Y 441.896,Z 989.03,A -85,B 0,C 180,E1 8461.957,E2 8461.957} C_VEL
LIN {X 0,Y 441.574,Z 989.03,A -85,B 0,C 180,E1 8467.857,E2 8467.857} C_VEL
LIN {X 0,Y 441.336,Z 989.03,A -85,B 0,C 180,E1 8473.847,E2 8473.847} C_VEL
LIN {X 0,Y 441.153,Z 989.03,A -85,B 0,C 180,E1 8480.002,E2 8480.002} C_VEL
LIN {X 0,Y 440.964,Z 989.03,A -85,B 0,C 180,E1 8486.414,E2 8486.414} C_VEL
LIN {X 0,Y 440.747,Z 989.03,A -85,B 0,C 180,E1 8493.215,E2 8493.215} C_VEL
LIN {X 0,Y 440.803,Z 989.03,A -85,B 0,C 180,E1 8498.064,E2 8498.064} C_VEL
LIN {X 0,Y 440.672,Z 989.03,A -85,B 0,C 180,E1 8504.023,E2 8504.023} C_VEL
LIN {X 0,Y 440.797,Z 989.031,A -85,B 0,C 180,E1 8506.344,E2 8506.344} C_VEL
LIN {X 0,Y 451.021,Z 1019.005,A -85,B 0,C 180,E1 8509.5,E2 8509.5} C_VEL
LIN {X 0,Y 464.611,Z 1046.627,A -85,B 0,C 180,E1 8511.29,E2 8511.29} C_VEL
LIN {X 0,Y 467.371,Z 1050.692,A -85,B 0,C 180,E1 8511.608,E2 8511.608} C_VEL
LIN {X 0,Y 465.043,Z 1093.315,A -85,B 0,C 180,E1 8512.793,E2 8512.793} C_VEL
LIN {X 0,Y 461.487,Z 1133.169,A -85,B 0,C 180,E1 8514.638,E2 8514.638} C_VEL
LIN {X 0,Y 457.596,Z 1168.105,A -85,B 0,C 180,E1 8516.952,E2 8516.952} C_VEL
LIN {X 0,Y 452.207,Z 1182.786,A -85,B 0,C 180,E1 8517.969,E2 8517.969} C_VEL
LIN {X 0,Y 446.664,Z 1196.79,A -85,B 0,C 180,E1 8519.099,E2 8519.099} C_VEL
LIN {X 0,Y 442.534,Z 1229.054,A -85,B 0,C 180,E1 8522.83,E2 8522.83} C_VEL
LIN {X 0,Y 438.86,Z 1257.771,A -85,B 0,C 180,E1 8527.246,E2 8527.246} C_VEL
LIN {X 0,Y 436.36,Z 1280.148,A -85,B 0,C 180,E1 8531.87,E2 8531.87} C_VEL
LIN {X 0,Y 434.9,Z 1296.846,A -85,B 0,C 180,E1 8536.655,E2 8536.655} C_VEL
LIN {X 0,Y 434.288,Z 1306.563,A -85,B 0,C 180,E1 8541.008,E2 8541.008} C_VEL
LIN {X 0,Y 434.016,Z 1312.922,A -85,B 0,C 180,E1 8546.016,E2 8546.016} C_VEL
LIN {X 0,Y 434.046,Z 1314.5,A -85,B 0,C 180,E1 8550.004,E2 8550.004} C_VEL
LIN {X 0,Y 434.013,Z 1312.925,A -85,B 0,C 180,E1 8553.991,E2 8553.991} C_VEL
LIN {X 0,Y 434.292,Z 1306.54,A -85,B 0,C 180,E1 8559,E2 8559} C_VEL
LIN {X 0,Y 435.076,Z 1294.785,A -85,B 0,C 180,E1 8564.055,E2 8564.055} C_VEL
LIN {X 0,Y 436.465,Z 1278.99,A -85,B 0,C 180,E1 8568.335,E2 8568.335} C_VEL
LIN {X 0,Y 438.872,Z 1256.245,A -85,B 0,C 180,E1 8572.761,E2 8572.761} C_VEL
LIN {X 0,Y 441.997,Z 1228.225,A -85,B 0,C 180,E1 8576.835,E2 8576.835} C_VEL
LIN {X 0,Y 445.61,Z 1195.388,A -85,B 0,C 180,E1 8580.384,E2 8580.384} C_VEL
LIN {X 0,Y 449.357,Z 1157.912,A -85,B 0,C 180,E1 8583.392,E2 8583.392} C_VEL
LIN {X 0,Y 452.925,Z 1116.245,A -85,B 0,C 180,E1 8585.794,E2 8585.794} C_VEL
LIN {X 0,Y 455.94,Z 1074.027,A -85,B 0,C 180,E1 8587.423,E2 8587.423} C_VEL
LIN {X 0,Y 456.446,Z 1050.754,A -85,B 0,C 180,E1 8588.074,E2 8588.074} C_VEL
LIN {X 0,Y 445.742,Z 1028.871,A -85,B 0,C 180,E1 8589.386,E2 8589.386} C_VEL
LIN {X 0,Y 435.223,Z 996.887,A -85,B 0,C 180,E1 8591.154,E2 8591.154} C_VEL
LIN {X 0,Y 432.944,Z 989.03,A -85,B 0,C 180,E1 8591.985,E2 8591.985} C_VEL
